    // Geometric and Coordinate Transformations
    node_F_VN_CalibrateCamera : Node_F_VN_CalibrateCamera;
    //node_F_VN_CalibrateCameraExp : Node_F_VN_CalibrateCameraExp;
    //node_F_VN_CalibrateCameraExp2 : Node_F_VN_CalibrateCameraExp2;
    //node_F_VN_CalibrateCameraExp3 : Node_F_VN_CalibrateCameraExp3;
    //node_F_VN_CalibrateCameraManually : Node_F_VN_CalibrateCameraManually;
    //node_F_VN_CalibrateCameraManuallyExp : Node_F_VN_CalibrateCameraManuallyExp;
    node_F_VN_CalibrateCameraPlanar : Node_F_VN_CalibrateCameraPlanar;
    //node_F_VN_CalibrateCameraPlanarExp : Node_F_VN_CalibrateCameraPlanarExp;
    //node_F_VN_CalibrateLinescanCamera : Node_F_VN_CalibrateLinescanCamera;
    //node_F_VN_CalibrateLinescanCameraExp : Node_F_VN_CalibrateLinescanCamera;
    node_F_VN_CompensateLensDistortion : Node_F_VN_CompensateLensDistortion;
    node_F_VN_CompensateLensDistortionExp1 : Node_F_VN_CompensateLensDistortionExp1;
    node_F_VN_CompensateLensDistortionExp2 : Node_F_VN_CompensateLensDistortionExp2;
    node_F_VN_CompensateLensDistortionForPoints : Node_F_VN_CompensateLensDistortionForPoints;
    node_F_VN_CompensateLensDistortionForPointsExp1 : Node_F_VN_CompensateLensDistortionForPointsExp1;
    node_F_VN_CompensateLensDistortionForPointsExp2 : Node_F_VN_CompensateLensDistortionForPointsExp2;
    node_F_VN_DetectPatternPoints : Node_F_VN_DetectPatternPoints;
    //node_F_VN_DetectPatternPointsExp : Node_F_VN_DetectPatternPointsExp;
    node_F_VN_GenerateCalibrationPatternReferencePoints : Node_F_VN_GenerateCalibrationPatternReferencePoints;
    //node_F_VN_ImagePointsWorldDistance : Node_F_VN_ImagePointsWorldDistance;
    node_F_VN_SolvePnP : Node_F_VN_SolvePnP;
    node_F_VN_SolvePnPExp : Node_F_VN_SolvePnPExp;
    node_F_VN_SortDetectedPatternPoints : Node_F_VN_SortDetectedPatternPoints;
    //node_F_VN_TransformCoordinatesImageToWorld_Container : Node_F_VN_TransformCoordinatesImageToWorld_Container;
    //node_F_VN_TransformCoordinatesImageToWorld_Point : Node_F_VN_TransformCoordinatesImageToWorld_Point;
    //node_F_VN_TransformCoordinatesPlanar_Container : Node_F_VN_TransformCoordinatesPlanar_Container;
    //node_F_VN_TransformCoordinatesPlanar_Point : Node_F_VN_TransformCoordinatesPlanar_Point;
    //node_F_VN_TransformCoordinatesWorldToImage_Container : Node_F_VN_TransformCoordinatesWorldToImage_Container;
    //node_F_VN_TransformCoordinatesWorldToImage_Point : Node_F_VN_TransformCoordinatesWorldToImage_Point;
    node_F_VN_AlignRotatedImageRegion : Node_F_VN_AlignRotatedImageRegion;
    node_F_VN_AlignRotatedImageRegionExp : Node_F_VN_AlignRotatedImageRegionExp;
    node_F_VN_ApplyRotationToAffineTransformation : Node_F_VN_ApplyRotationToAffineTransformation;
    node_F_VN_ApplyRotationToAffineTransformationExp : Node_F_VN_ApplyRotationToAffineTransformationExp;
    node_F_VN_ApplyScalingToAffineTransformation : Node_F_VN_ApplyScalingToAffineTransformation;
    node_F_VN_ApplyScalingToAffineTransformationExp : Node_F_VN_ApplyScalingToAffineTransformationExp;
    node_F_VN_ApplyTranslationToAffineTransformation : Node_F_VN_ApplyTranslationToAffineTransformation;
    node_F_VN_ApplyTranslationToAffineTransformationExp : Node_F_VN_ApplyTranslationToAffineTransformationExp;
    node_F_VN_ApplyYAxisInversionToAffineTransformation : Node_F_VN_ApplyYAxisInversionToAffineTransformation;
    node_F_VN_ApplyYAxisInversionToAffineTransformationExp : Node_F_VN_ApplyYAxisInversionToAffineTransformationExp;
    // Polarization
    node_F_VN_DemosaicPolarizedImage : Node_F_VN_DemosaicPolarizedImage;
    node_F_VN_AngleAndDegreeOfLinearPolarization : Node_F_VN_AngleAndDegreeOfLinearPolarization;
    node_F_VN_PolarizedImageGlareReduction : Node_F_VN_PolarizedImageGlareReduction;
    node_F_VN_ConvertCartesianToPolarAngleImage : Node_F_VN_ConvertCartesianToPolarAngleImage;
    node_F_VN_ConvertCartesianToPolarAngleImageExp : Node_F_VN_ConvertCartesianToPolarAngleImageExp;
    node_F_VN_ConvertCartesianToPolarAngles : Node_F_VN_ConvertCartesianToPolarAngles;
    node_F_VN_ConvertCartesianToPolarAnglesExp : Node_F_VN_ConvertCartesianToPolarAnglesExp;
    node_F_VN_ConvertCartesianToPolarImages : Node_F_VN_ConvertCartesianToPolarImages;
    node_F_VN_ConvertCartesianToPolarImagesExp : Node_F_VN_ConvertCartesianToPolarImagesExp;
    node_F_VN_ConvertCartesianToPolarMagnitudeImage : Node_F_VN_ConvertCartesianToPolarMagnitudeImage;
    node_F_VN_ConvertCartesianToPolarMagnitudes : Node_F_VN_ConvertCartesianToPolarMagnitudes;
    node_F_VN_ConvertCartesianToPolarPoints : Node_F_VN_ConvertCartesianToPolarPoints;
    node_F_VN_ConvertCartesianToPolarPointsExp : Node_F_VN_ConvertCartesianToPolarPointsExp;
    node_F_VN_ConvertPolarToCartesianImages : Node_F_VN_ConvertPolarToCartesianImages;
    node_F_VN_ConvertPolarToCartesianImagesExp : Node_F_VN_ConvertPolarToCartesianImagesExp;
    node_F_VN_ConvertPolarToCartesianPoints : Node_F_VN_ConvertPolarToCartesianPoints;
    node_F_VN_ConvertPolarToCartesianPointsExp : Node_F_VN_ConvertPolarToCartesianPointsExp;
    //node_F_VN_DecomposeAffineTransformation : F_VN_DecomposeAffineTransformation;
    node_F_VN_DecomposeAffineTransformation : Node_F_VN_DecomposeAffineTransformation;
    node_F_VN_DecomposeAffineTransformationExp : Node_F_VN_DecomposeAffineTransformationExp;
    //node_F_VN_DecomposeHomography : Node_F_VN_DecomposeHomography;
    //node_F_VN_DecomposeHomographyExp : Node_F_VN_DecomposeHomographyExp;
    node_F_VN_FlipImage : Node_F_VN_FlipImage;
    node_F_VN_GenerateAffineTransformationUnitMatrix2D : Node_F_VN_GenerateAffineTransformationUnitMatrix2D;
    node_F_VN_GetAffineTransformation : Node_F_VN_GetAffineTransformation;
    node_F_VN_GetAffineTransformation2D : Node_F_VN_GetAffineTransformation2D;
    //node_F_VN_GetAffineTransformation2DExp : Node_F_VN_GetAffineTransformation2DExp;
    node_F_VN_GetPerspectiveTransformation : Node_F_VN_GetPerspectiveTransformation;
    node_F_VN_Homography : Node_F_VN_Homography;
    node_F_VN_HomographyExp : Node_F_VN_HomographyExp;
    node_F_VN_InvertAffineTransformation : Node_F_VN_InvertAffineTransformation;
    node_F_VN_PerspectiveTransformation : Node_F_VN_PerspectiveTransformation;
    node_F_VN_PyramidDown : Node_F_VN_PyramidDown;
    node_F_VN_PyramidUp : Node_F_VN_PyramidUp;
    node_F_VN_ConvertMaps : Node_F_VN_ConvertMaps;
    node_F_VN_RemapImage : Node_F_VN_RemapImage;
    node_F_VN_RemapImageExp : Node_F_VN_RemapImageExp;
    node_F_VN_RemapImageToLogPolarSpace : Node_F_VN_RemapImageToLogPolarSpace;
    node_F_VN_RemapImageToLogPolarSpaceExp : Node_F_VN_RemapImageToLogPolarSpaceExp;
    node_F_VN_RemapImageToLogPolarSpaceExp2 : Node_F_VN_RemapImageToLogPolarSpaceExp2;
    node_F_VN_RemapImageToPolarSpace : Node_F_VN_RemapImageToPolarSpace;
    node_F_VN_RemapImageToPolarSpaceExp : Node_F_VN_RemapImageToPolarSpaceExp;
    node_F_VN_RemapImageToPolarSpaceExp2 : Node_F_VN_RemapImageToPolarSpaceExp2;
    node_F_VN_ResizeImage : Node_F_VN_ResizeImage;
    node_F_VN_ResizeImageExp : Node_F_VN_ResizeImageExp;
	node_F_VN_ResizeRegion_TcVnRectangle_DINT : Node_F_VN_ResizeRegion_TcVnRectangle_DINT;
    node_F_VN_RotateImage : Node_F_VN_RotateImage;
    node_F_VN_RotateImageExp : Node_F_VN_RotateImageExp;
    node_F_VN_RotateImageExp2 : Node_F_VN_RotateImageExp2;
    node_F_VN_WarpAffine : Node_F_VN_WarpAffine;
    node_F_VN_WarpAffine_Container : Node_F_VN_WarpAffine_Container;
    node_F_VN_WarpAffine_Point : Node_F_VN_WarpAffine_Point;
    node_F_VN_WarpAffine_Rectangle : Node_F_VN_WarpAffine_Rectangle;
    node_F_VN_WarpAffineExp : Node_F_VN_WarpAffineExp;
    node_F_VN_WarpPerspective : Node_F_VN_WarpPerspective;
    node_F_VN_WarpPerspective_Container : Node_F_VN_WarpPerspective_Container;
    node_F_VN_WarpPerspective_Point : Node_F_VN_WarpPerspective_Point;
    node_F_VN_WarpPerspective_Rectangle : Node_F_VN_WarpPerspective_Rectangle;
    node_F_VN_WarpPerspectiveExp : Node_F_VN_WarpPerspectiveExp;
    
	// Helpers
	node_Mux10Way_ITcVnImage : Node_Mux10Way_ITcVnImage;
	
    // Image Analysis
    //node_F_VN_AdjustActiveContour : Node_F_VN_AdjustActiveContour;
    node_F_VN_SalientFeatures : Node_F_VN_SalientFeatures;
    node_F_VN_FindRois : Node_F_VN_FindRois;
    node_F_VN_MergeRegions : Node_F_VN_MergeRegions;
    node_F_VN_DetectBlobs : Node_F_VN_DetectBlobs;
    node_F_VN_DetectBlobsExp : Node_F_VN_DetectBlobsExp;
    node_F_VN_FindContourHierarchyExp : Node_F_VN_FindContourHierarchyExp;
    node_F_VN_FindContours : Node_F_VN_FindContours;
    node_F_VN_FindContoursExp : Node_F_VN_FindContoursExp;
	node_F_VN_FindTemplateWalsh : Node_F_VN_FindTemplateWalsh;
	node_F_VN_FindTemplateWalsh_AngleRange : Node_F_VN_FindTemplateWalsh_AngleRange;
	node_F_VN_FindTemplateWalshExp : Node_F_VN_FindTemplateWalshExp;
	node_F_VN_FindTemplateWalshExp_AngleRange : Node_F_VN_FindTemplateWalshExp_AngleRange;
    node_F_VN_HoughCircles : Node_F_VN_HoughCircles;
    node_F_VN_HoughCirclesExp : Node_F_VN_HoughCirclesExp;
    node_F_VN_HoughLines : Node_F_VN_HoughLines;
    //node_F_VN_HoughLinesExp : Node_F_VN_HoughLinesExp;
    node_F_VN_HoughLinesP : Node_F_VN_HoughLinesP;
    node_F_VN_HoughLinesPExp : Node_F_VN_HoughLinesPExp;
    node_F_VN_MatchImageHuMoments : Node_F_VN_MatchImageHuMoments;
    node_F_VN_MatchTemplate : Node_F_VN_MatchTemplate;
    node_F_VN_MatchTemplateAndEvaluate : Node_F_VN_MatchTemplateAndEvaluate;
	node_F_VN_MatchTemplateWalsh : Node_F_VN_MatchTemplateWalsh;
	node_F_VN_MatchTemplateWalshExp : Node_F_VN_MatchTemplateWalshExp;
    node_F_VN_MatchTemplateAndEvaluateExp : Node_F_VN_MatchTemplateAndEvaluateExp;
    node_F_VN_MatchTemplateExp : Node_F_VN_MatchTemplateExp;
    node_F_VN_CannyEdgeDetection : Node_F_VN_CannyEdgeDetection;
    node_F_VN_CannyEdgeDetectionExp : Node_F_VN_CannyEdgeDetectionExp;
    node_F_VN_ConnectedComponents : Node_F_VN_ConnectedComponents;
    node_F_VN_ConnectedComponentsExp : Node_F_VN_ConnectedComponentsExp;
    node_F_VN_ConnectedComponentsWithStats : Node_F_VN_ConnectedComponentsWithStats;
    node_F_VN_ConnectedComponentsWithStatsExp : Node_F_VN_ConnectedComponentsWithStatsExp;
    node_F_VN_CountNonZeroPixels : Node_F_VN_CountNonZeroPixels;
    node_F_VN_DistanceTransformation : Node_F_VN_DistanceTransformation;
    node_F_VN_DistanceTransformationExp : Node_F_VN_DistanceTransformationExp;
    node_F_VN_GetConnectedComponent : Node_F_VN_GetConnectedComponent;
    node_F_VN_GetConnectedComponentExp : Node_F_VN_GetConnectedComponentExp;
    node_F_VN_ImageAverage : Node_F_VN_ImageAverage;
    node_F_VN_ImageAverageExp : Node_F_VN_ImageAverageExp;
    node_F_VN_ImageAverageStdDev : Node_F_VN_ImageAverageStdDev;
    node_F_VN_ImageAverageStdDevExp : Node_F_VN_ImageAverageStdDevExp;
    node_F_VN_ImageCenterOfMass : Node_F_VN_ImageCenterOfMass;
    node_F_VN_ImageCenterOfMassExp : Node_F_VN_ImageCenterOfMassExp;
    node_F_VN_ImageMedian : Node_F_VN_ImageMedian;
    node_F_VN_ImageMedianExp : Node_F_VN_ImageMedianExp;
    node_F_VN_ImageMoments : Node_F_VN_ImageMoments;
    node_F_VN_MaxPixelValue : Node_F_VN_MaxPixelValue;
    node_F_VN_MaxPixelValueExp : Node_F_VN_MaxPixelValueExp;
    node_F_VN_MinPixelValue : Node_F_VN_MinPixelValue;
    node_F_VN_MinPixelValueExp : Node_F_VN_MinPixelValueExp;
    node_F_VN_RegionOrientation : Node_F_VN_RegionOrientation;
    node_F_VN_RegionOrientationExp : Node_F_VN_RegionOrientationExp;
    node_F_VN_ImageAbsoluteAverage : Node_F_VN_ImageAbsoluteAverage;
    node_F_VN_UprightInnerRectangle : Node_F_VN_UprightInnerRectangle;
    node_F_VN_UprightInnerRectangleExp : Node_F_VN_UprightInnerRectangleExp;
    
    // Image Color and Contrast Processing
    node_F_VN_ApplyColorMap : Node_F_VN_ApplyColorMap;
    //node_F_VN_ApplyLut : Node_F_VN_ApplyLut;
    node_F_VN_Clahe : Node_F_VN_Clahe;
    node_F_VN_ClaheExp : Node_F_VN_ClaheExp;
    node_F_VN_ConvertColorSpace : Node_F_VN_ConvertColorSpace;
    node_F_VN_GenerateColorMap : Node_F_VN_GenerateColorMap;
    node_F_VN_GenerateCustomColorMap : Node_F_VN_GenerateCustomColorMap;
    node_F_VN_Histogram : Node_F_VN_Histogram;
    node_F_VN_HistogramEqualization : Node_F_VN_HistogramEqualization;
    node_F_VN_HistogramEqualizationExp : Node_F_VN_HistogramEqualizationExp;
	node_F_VN_HistogramExp : Node_F_VN_HistogramExp;
    node_F_VN_InvertImageColor : Node_F_VN_InvertImageColor;
    node_F_VN_InvertImageColorExp : Node_F_VN_InvertImageColorExp;
    node_F_VN_NormalizeImage : Node_F_VN_NormalizeImage;
    node_F_VN_NormalizeImageExp : Node_F_VN_NormalizeImageExp;
    node_F_VN_NormalizeImageForDisplay : Node_F_VN_NormalizeImageForDisplay;
    //node_F_VN_ReferenceColorSimilarity_ITcVnColorModel : Node_F_VN_ReferenceColorSimilarity_ITcVnColorModel;
    //node_F_VN_ReferenceColorSimilarity_ITcVnMlModel : Node_F_VN_ReferenceColorSimilarity_ITcVnMlModel;
    node_F_VN_ReferenceColorSimilarity_TcVnVector3_LREAL : Node_F_VN_ReferenceColorSimilarity_TcVnVector3_LREAL;
    //node_F_VN_ReferenceColorSimilarityExp_ITcVnColorModel : Node_F_VN_ReferenceColorSimilarityExp_ITcVnColorModel;
    //node_F_VN_ReferenceColorSimilarityExp_ITcVnColorModel : Node_F_VN_ReferenceColorSimilarityExp_ITcVnColorModel;
    node_F_VN_ReferenceColorSimilarityExp_TcVnVector3_LREAL : Node_F_VN_ReferenceColorSimilarityExp_TcVnVector3_LREAL;
    //node_F_VN_TrainImageColor : Node_F_VN_TrainImageColor;
    //node_F_VN_TrainImageColor_ITcVnMlModel : Node_F_VN_TrainImageColor_ITcVnMlModel;
    //node_F_VN_TrainImageColorExp : Node_F_VN_TrainImageColorExp;
    //node_F_VN_TrainImageColorExp_ITcVnMlModel : Node_F_VN_TrainImageColorExp_ITcVnMlModel;
    //node_F_VN_TrainImageColorExp2 : Node_F_VN_TrainImageColorExp2;
    //node_F_VN_TrainImageColorExp2_ITcVnMlModel : Node_F_VN_TrainImageColorExp2_ITcVnMlModel;
    node_F_VN_WhiteBalance : Node_F_VN_WhiteBalance;
    
    // Image Filtering
    node_F_VN_BilateralFilter : Node_F_VN_BilateralFilter;
    node_F_VN_BilateralFilterExp : Node_F_VN_BilateralFilterExp;
    node_F_VN_BoxFilter : Node_F_VN_BoxFilter;
    node_F_VN_BoxFilterExp : Node_F_VN_BoxFilterExp;
    node_F_VN_BrightBorderObjects : Node_F_VN_BrightBorderObjects;
    node_F_VN_CreateStructuringElement : Node_F_VN_CreateStructuringElement;
    //node_F_VN_CustomFilter : Node_F_VN_CustomFilter;
    //node_F_VN_CustomFilterExp : Node_F_VN_CustomFilterExp;
    node_F_VN_DarkBorderObjects : Node_F_VN_DarkBorderObjects;
    node_F_VN_FillHoles : Node_F_VN_FillHoles;
    node_F_VN_GaussianFilter : Node_F_VN_GaussianFilter;
    node_F_VN_GaussianFilterExp : Node_F_VN_GaussianFilterExp;
    node_F_VN_LaplacianFilter : Node_F_VN_LaplacianFilter;
    node_F_VN_LaplacianFilterExp : Node_F_VN_LaplacianFilterExp;
    node_F_VN_LocalMaxima : Node_F_VN_LocalMaxima;
    node_F_VN_LocalMinima : Node_F_VN_LocalMinima;
    node_F_VN_MedianFilter : Node_F_VN_MedianFilter;
    node_F_VN_MorphologicalOperator : Node_F_VN_MorphologicalOperator;
    node_F_VN_RemoveLocalMaxima : Node_F_VN_RemoveLocalMaxima;
    node_F_VN_RemoveLocalMinima : Node_F_VN_RemoveLocalMinima;
    node_F_VN_ScharrFilter : Node_F_VN_ScharrFilter;
    node_F_VN_ScharrFilterExp : Node_F_VN_ScharrFilterExp;
    //node_F_VN_SeparableCustomFilter : Node_F_VN_SeparableCustomFilter;
    //node_F_VN_SeparableCustomFilterExp : Node_F_VN_SeparableCustomFilterExp;
    node_F_VN_SobelFilter : Node_F_VN_SobelFilter;
    node_F_VN_SobelFilterExp : Node_F_VN_SobelFilterExp;
    node_F_VN_VarianceFilter : Node_F_VN_VarianceFilter;
    node_F_VN_VarianceFilterExp : Node_F_VN_VarianceFilterExp;
    
    // Image Segmentation
    node_F_VN_AdaptiveThreshold : Node_F_VN_AdaptiveThreshold;
    node_F_VN_AdaptiveThresholdExp : Node_F_VN_AdaptiveThresholdExp;
    node_F_VN_CheckColorRange : Node_F_VN_CheckColorRange;
    node_F_VN_DoubleThreshold : Node_F_VN_DoubleThreshold;
    node_F_VN_Threshold : Node_F_VN_Threshold;
    node_F_VN_WatershedSegmentationExp : Node_F_VN_WatershedSegmentationExp;
    node_F_VN_SauvolaThreshold : Node_F_VN_SauvolaThreshold;
    
    // Keypoint Features
    node_F_VN_FilterGoodMatches : Node_F_VN_FilterGoodMatches;
    node_F_VN_FindReferenceKeyPointsInImage : Node_F_VN_FindReferenceKeyPointsInImage;
    node_F_VN_FindReferenceKeyPointsInImageAKAZE : Node_F_VN_FindReferenceKeyPointsInImageAKAZE;
    node_F_VN_FindReferenceKeyPointsInImageAKAZEExp : Node_F_VN_FindReferenceKeyPointsInImageAKAZEExp;
    node_F_VN_FindReferenceKeyPointsInImageBRISK : Node_F_VN_FindReferenceKeyPointsInImageBRISK;
    node_F_VN_FindReferenceKeyPointsInImageBRISKExp : Node_F_VN_FindReferenceKeyPointsInImageBRISKExp;
    node_F_VN_FindReferenceKeyPointsInImageExp : Node_F_VN_FindReferenceKeyPointsInImageExp;
    node_F_VN_FindReferenceKeyPointsInImageORB : Node_F_VN_FindReferenceKeyPointsInImageORB;
    node_F_VN_FindReferenceKeyPointsInImageORBExp : Node_F_VN_FindReferenceKeyPointsInImageORBExp;
    node_F_VN_GetMatchCoordinates : Node_F_VN_GetMatchCoordinates;
    node_F_VN_KeyPointsAGAST : Node_F_VN_KeyPointsAGAST;
    node_F_VN_KeyPointsAGASTExp : Node_F_VN_KeyPointsAGASTExp;
    node_F_VN_KeyPointsAndDescriptorsAKAZE : Node_F_VN_KeyPointsAndDescriptorsAKAZE;
    node_F_VN_KeyPointsAndDescriptorsAKAZEExp : Node_F_VN_KeyPointsAndDescriptorsAKAZEExp;
    node_F_VN_KeyPointsAndDescriptorsBRISK : Node_F_VN_KeyPointsAndDescriptorsBRISK;
    node_F_VN_KeyPointsAndDescriptorsBRISKExp : Node_F_VN_KeyPointsAndDescriptorsBRISKExp;
    node_F_VN_KeyPointsAndDescriptorsKAZE : Node_F_VN_KeyPointsAndDescriptorsKAZE;
    node_F_VN_KeyPointsAndDescriptorsKAZEExp : Node_F_VN_KeyPointsAndDescriptorsKAZEExp;
    node_F_VN_KeyPointsAndDescriptorsORB : Node_F_VN_KeyPointsAndDescriptorsORB;
    node_F_VN_KeyPointsAndDescriptorsORBExp : Node_F_VN_KeyPointsAndDescriptorsORBExp;
    node_F_VN_KeyPointsFAST : Node_F_VN_KeyPointsFAST;
    node_F_VN_KeyPointsFASTExp : Node_F_VN_KeyPointsFASTExp;
    node_F_VN_KeyPointsGFTT : Node_F_VN_KeyPointsGFTT;
    node_F_VN_KeyPointsGFTTExp : Node_F_VN_KeyPointsGFTTExp;
    node_F_VN_KeyPointsMSER : Node_F_VN_KeyPointsMSER;
    node_F_VN_KeyPointsMSERExp : Node_F_VN_KeyPointsMSERExp;
    node_F_VN_KeyPointsSB : Node_F_VN_KeyPointsSB;
    node_F_VN_KeyPointsSBExp : Node_F_VN_KeyPointsSBExp;
    node_F_VN_MatchDescriptorsBF : Node_F_VN_MatchDescriptorsBF;
    node_F_VN_MatchDescriptorsBFExp : Node_F_VN_MatchDescriptorsBFExp;
    node_F_VN_MatchDescriptorsFlannLsh : Node_F_VN_MatchDescriptorsFlannLsh;
    node_F_VN_MatchDescriptorsFlannLshExp : Node_F_VN_MatchDescriptorsFlannLshExp;
    node_F_VN_MatchDescriptorsKnnBF : Node_F_VN_MatchDescriptorsKnnBF;
    node_F_VN_MatchDescriptorsKnnBFExp : Node_F_VN_MatchDescriptorsKnnBFExp;
    node_F_VN_MatchDescriptorsKnnFlannLsh : Node_F_VN_MatchDescriptorsKnnFlannLsh;
    node_F_VN_MatchDescriptorsKnnFlannLshExp : Node_F_VN_MatchDescriptorsKnnFlannLshExp;
    node_F_VN_RegionsMSER : Node_F_VN_RegionsMSER;
    node_F_VN_RegionsMSERExp : Node_F_VN_RegionsMSERExp;
    
    // Machine Learning
    //node_F_VN_CreateBoostClassifier : Node_F_VN_CreateBoostClassifier;
    //node_F_VN_CreateBoostClassifierExp : Node_F_VN_CreateBoostClassifierExp;
    //node_F_VN_CreateBoostClassifierExp2 : Node_F_VN_CreateBoostClassifierExp2;
    //node_F_VN_CreateKmppModel : Node_F_VN_CreateKmppModel;
    //node_F_VN_CreateKmppModelExp : Node_F_VN_CreateKmppModelExp;
    //node_F_VN_CreateKnnModel : Node_F_VN_CreateKnnModel;
    //node_F_VN_CreateLbgModel : Node_F_VN_CreateLbgModel;
    //node_F_VN_CreateLbgModelExp : Node_F_VN_CreateLbgModelExp;
    //node_F_VN_CreateLdaTransform : Node_F_VN_CreateLdaTransform;
    //node_F_VN_CreateLdaTransformViaComponentNum : Node_F_VN_CreateLdaTransformViaComponentNum;
    //node_F_VN_CreateNbcModel : Node_F_VN_CreateNbcModel;
    //node_F_VN_CreatePcaTransform : Node_F_VN_CreatePcaTransform;
    //node_F_VN_CreatePcaTransformViaComponentNum : Node_F_VN_CreatePcaTransformViaComponentNum;
    //node_F_VN_CreatePcaTransformViaVariance : Node_F_VN_CreatePcaTransformViaVariance;
    //node_F_VN_CreateRTreesModel : Node_F_VN_CreateRTreesModel;
    //node_F_VN_CreateRTreesModelExp : Node_F_VN_CreateRTreesModelExp;
    //node_F_VN_CreateRTreesModelExp2 : Node_F_VN_CreateRTreesModelExp2;
    //node_F_VN_CreateStaModel : Node_F_VN_CreateStaModel;
    //node_F_VN_CreateStaModelExp : Node_F_VN_CreateStaModelExp;
    //node_F_VN_CreateStaModelExp2 : Node_F_VN_CreateStaModelExp2;
    //node_F_VN_CreateSvmModel : Node_F_VN_CreateSvmModel;
    //node_F_VN_CreateSvmModelExp : Node_F_VN_CreateSvmModelExp;
    //node_F_VN_CreateSvmModelExp2 : Node_F_VN_CreateSvmModelExp2;
    //node_F_VN_CreateSvmSgdClassifier : Node_F_VN_CreateSvmSgdClassifier;
    //node_F_VN_CreateSvmSgdClassifierExp : Node_F_VN_CreateSvmSgdClassifierExp;
    //node_F_VN_FeatureScaling : Node_F_VN_FeatureScaling;
    //node_F_VN_FeatureScalingExp : Node_F_VN_FeatureScalingExp;
    //node_F_VN_FeatureTransform : Node_F_VN_FeatureTransform;
    //node_F_VN_GetBatchClusters : Node_F_VN_GetBatchClusters;
    //node_F_VN_GetBatchClustersExp : Node_F_VN_GetBatchClustersExp;
    //node_F_VN_GetBatchNovelties : Node_F_VN_GetBatchNovelties;
    //node_F_VN_GetClusterCenter : Node_F_VN_GetClusterCenter;
    //node_F_VN_GetClusterNum : Node_F_VN_GetClusterNum;
    //node_F_VN_GetFeatureScales : Node_F_VN_GetFeatureScales;
    //node_F_VN_GetSampleCluster : Node_F_VN_GetSampleCluster;
    //node_F_VN_GetSampleClusterExp : Node_F_VN_GetSampleClusterExp;
    //node_F_VN_GetSampleNovelty : Node_F_VN_GetSampleNovelty;
    //node_F_VN_InverseFeatureScaling : Node_F_VN_InverseFeatureScaling;
    //node_F_VN_InverseFeatureScaling_REAL : Node_F_VN_InverseFeatureScaling_REAL;
    //node_F_VN_InverseFeatureScalingExp : Node_F_VN_InverseFeatureScalingExp;
    //node_F_VN_InverseFeatureScalingExp_REAL : Node_F_VN_InverseFeatureScalingExp_REAL;
    //node_F_VN_InverseFeatureTransform : Node_F_VN_InverseFeatureTransform;
    //node_F_VN_PredictBatch : Node_F_VN_PredictBatch;
    //node_F_VN_PredictBatchExp : Node_F_VN_PredictBatchExp;
    //node_F_VN_PredictSampleClass : Node_F_VN_PredictSampleClass;
    //node_F_VN_PredictSampleClassExp : Node_F_VN_PredictSampleClassExp;
    //node_F_VN_PredictSampleScalar : Node_F_VN_PredictSampleScalar;
    //node_F_VN_PredictSampleScalarExp : Node_F_VN_PredictSampleScalarExp;
    //node_F_VN_PredictSampleVector : Node_F_VN_PredictSampleVector;
    //node_F_VN_PredictSampleVectorExp : Node_F_VN_PredictSampleVectorExp;
    //node_F_VN_TrainBatch : Node_F_VN_TrainBatch;
    //node_F_VN_TrainBatchClusters : Node_F_VN_TrainBatchClusters;
    //node_F_VN_TrainSample : Node_F_VN_TrainSample;
    //node_F_VN_TrainSampleClass : Node_F_VN_TrainSampleClass;
    //node_F_VN_TrainSampleCluster : Node_F_VN_TrainSampleCluster;
    //node_F_VN_TrainSampleScalar : Node_F_VN_TrainSampleScalar;
    //node_F_VN_TrainSampleVector : Node_F_VN_TrainSampleVector;

    // Measurement
    node_F_VN_AdjustSearchWindowOrientationToLinearEdge : Node_F_VN_AdjustSearchWindowOrientationToLinearEdge;
	node_F_VN_ClosestPointsBF : Node_F_VN_ClosestPointsBF;
    node_F_VN_LocateAxisAlignedEdges : Node_F_VN_LocateAxisAlignedEdges;
    node_F_VN_LocateAxisAlignedEdgesExp : Node_F_VN_LocateAxisAlignedEdgesExp;
	node_F_VN_LocateCircularArc : Node_F_VN_LocateCircularArc;
    node_F_VN_LocateCircularArcExp : Node_F_VN_LocateCircularArcExp;
    node_F_VN_LocateCircularArcExp2 : Node_F_VN_LocateCircularArcExp2;
    node_F_VN_LocateEdge : Node_F_VN_LocateEdge;
    node_F_VN_LocateEdgeExp : Node_F_VN_LocateEdgeExp;
    node_F_VN_LocateEdgeExp2 : Node_F_VN_LocateEdgeExp2;
    node_F_VN_LocateEdges : Node_F_VN_LocateEdges;
    node_F_VN_LocateEdgesExp : Node_F_VN_LocateEdgesExp;
    node_F_VN_LocateEdgesExp2 : Node_F_VN_LocateEdgesExp2;
    node_F_VN_LocateEllipse : Node_F_VN_LocateEllipse;
	node_F_VN_LocateEllipseExp : Node_F_VN_LocateEllipseExp;
    node_F_VN_LocateEllipseExp2 : Node_F_VN_LocateEllipseExp2;
    node_F_VN_MeasureAngleBetweenEdges : Node_F_VN_MeasureAngleBetweenEdges;
    node_F_VN_MeasureAngleBetweenEdgesExp : Node_F_VN_MeasureAngleBetweenEdgesExp;
    node_F_VN_MeasureAngleBetweenEdgesExp2 : Node_F_VN_MeasureAngleBetweenEdgesExp2;
    node_F_VN_MeasureEdgeDistance : Node_F_VN_MeasureEdgeDistance;
	node_F_VN_MeasureEdgeDistanceExp : Node_F_VN_MeasureEdgeDistanceExp;
    node_F_VN_MeasureEdgeDistanceExp2 : Node_F_VN_MeasureEdgeDistanceExp2;
    node_F_VN_MeasureMinEdgeDistance : Node_F_VN_MeasureMinEdgeDistance;
    node_F_VN_MeasureMinEdgeDistanceExp : Node_F_VN_MeasureMinEdgeDistanceExp;
    node_F_VN_MeasureMinEdgeDistanceExp2 : Node_F_VN_MeasureMinEdgeDistanceExp2;
    
    // Miscellaneous
    node_F_VN_CheckFunctionInitialization : Node_F_VN_CheckFunctionInitialization;
    node_F_VN_ClipLineToBoundary : Node_F_VN_ClipLineToBoundary;
    node_F_VN_ClipLineToBoundary_ITcVnImage : Node_F_VN_ClipLineToBoundary_ITcVnImage;
    node_F_VN_ClipLineToBoundary_TcVnRectangle_DINT : Node_F_VN_ClipLineToBoundary_TcVnRectangle_DINT;
    //node_F_VN_ConvertITcUnknownToITcVnBitmapExport : Node_F_VN_ConvertITcUnknownToITcVnBitmapExport;
    //node_F_VN_ConvertITcUnknownToITcVnContainer : Node_F_VN_ConvertITcUnknownToITcVnContainer;
    //node_F_VN_ConvertITcUnknownToITcVnImage : Node_F_VN_ConvertITcUnknownToITcVnImage;
    //node_F_VN_ConvertITcUnknownToITcVnMlModel : Node_F_VN_ConvertITcUnknownToITcVnMlModel;
    node_F_VN_DeinitializeFunction : Node_F_VN_DeinitializeFunction;
    //node_F_VN_GetTimestamp : Node_F_VN_GetTimestamp;
    node_F_VN_HuMomentInvariants : Node_F_VN_HuMomentInvariants;
    //node_F_VN_InitMatrixStruct : Node_F_VN_InitMatrixStruct;
    node_F_VN_InvertMatrix3x3 : Node_F_VN_InvertMatrix3x3;
    node_F_VN_LineIntersectionPoint : Node_F_VN_LineIntersectionPoint;
    node_F_VN_LineIntersectionPointAndAngle : Node_F_VN_LineIntersectionPointAndAngle;
    //node_F_VN_MultiplyMatrices : Node_F_VN_MultiplyMatrices;
    node_F_VN_OrthogonalVector_TcVnVector2_DINT : Node_F_VN_OrthogonalVector_TcVnVector2_DINT;
    node_F_VN_OrthogonalVector_TcVnVector2_LREAL : Node_F_VN_OrthogonalVector_TcVnVector2_LREAL;
    node_F_VN_OrthogonalVector_TcVnVector2_REAL : Node_F_VN_OrthogonalVector_TcVnVector2_REAL;
    node_F_VN_PointToLineDistance_TcVnPoint2_DINT : Node_F_VN_PointToLineDistance_TcVnPoint2_DINT;
    node_F_VN_PointToLineDistance_TcVnPoint2_LREAL : Node_F_VN_PointToLineDistance_TcVnPoint2_LREAL;
    node_F_VN_PointToLineDistance_TcVnPoint2_REAL : Node_F_VN_PointToLineDistance_TcVnPoint2_REAL;
    node_F_VN_PointToPointDirection_TcVnPoint2_DINT : Node_F_VN_PointToPointDirection_TcVnPoint2_DINT;
    node_F_VN_PointToPointDirection_TcVnPoint2_LREAL : Node_F_VN_PointToPointDirection_TcVnPoint2_LREAL;
    node_F_VN_PointToPointDirection_TcVnPoint2_REAL : Node_F_VN_PointToPointDirection_TcVnPoint2_REAL;
    node_F_VN_PointToPointDistance_TcVnPoint2_DINT : Node_F_VN_PointToPointDistance_TcVnPoint2_DINT;
    node_F_VN_PointToPointDistance_TcVnPoint2_LREAL : Node_F_VN_PointToPointDistance_TcVnPoint2_LREAL;
    node_F_VN_PointToPointDistance_TcVnPoint2_REAL : Node_F_VN_PointToPointDistance_TcVnPoint2_REAL;
    node_F_VN_RotatedRectangleCorners : Node_F_VN_RotatedRectangleCorners;
    node_F_VN_RotatedRectangleIntersection : Node_F_VN_RotatedRectangleIntersection;
    //node_F_VN_SetRngSeed : Node_F_VN_SetRngSeed;
    //node_F_VN_UpdateTimestamp : Node_F_VN_UpdateTimestamp;
    
//     node_FB_VN_InitializeFunction : Node_FB_VN_InitializeFunction;
    
    // OCR
    node_F_VN_OCR : Node_F_VN_OCR;
    node_F_VN_OCRExp : Node_F_VN_OCRExp;
    
    // Texture Analysis
    node_F_VN_Granulometry : Node_F_VN_Granulometry;
    node_F_VN_HaralickFeatures : Node_F_VN_HaralickFeatures;
    
    // Neural Network
    //node_F_VN_ConvertDataLayout : Node_F_VN_ConvertDataLayout;
    //node_F_VN_ExecuteNeuralNetwork : Node_F_VN_ExecuteNeuralNetwork;
    //node_F_VN_ExecuteNeuralNetwork_MultiLayerOutput : Node_F_VN_ExecuteNeuralNetwork_MultiLayerOutput;
    //node_F_VN_ExecuteNeuralNetwork_SingleLayerOutput : Node_F_VN_ExecuteNeuralNetwork_SingleLayerOutput;
    //node_F_VN_GetNeuralNetworkLayerNames : Node_F_VN_GetNeuralNetworkLayerNames;
    //node_F_VN_NonMaxSuppression : Node_F_VN_NonMaxSuppression;
    //node_F_VN_NonMaxSuppressionExp : Node_F_VN_NonMaxSuppressionExp;
	node_F_VN_Reduce : Node_F_VN_Reduce;
	node_F_VN_ReduceArg : Node_F_VN_ReduceArg;
    //node_F_VN_ReshapeImage : Node_F_VN_ReshapeImage;
	node_F_VN_Sigmoid : Node_F_VN_Sigmoid;
	node_F_VN_SigmoidExp : Node_F_VN_SigmoidExp;
	node_F_VN_SoftMax : Node_F_VN_SoftMax;
	
END_VAR

METHOD PUBLIC RegisterWithNodeFactory
VAR_INPUT
	NodeFactory : I_NodeFactory;
END_VAR
// Algebraic Container Operations
NodeFactory.AddNodeAsPrototype('Vision/Algebraic Container Operations/F_VN_AddToContainerElements/F_VN_AddToContainerElements_DINT', node_F_VN_AddToContainerElements_DINT);
NodeFactory.AddNodeAsPrototype('Vision/Algebraic Container Operations/F_VN_AddToContainerElements/F_VN_AddToContainerElements_INT', node_F_VN_AddToContainerElements_INT);
NodeFactory.AddNodeAsPrototype('Vision/Algebraic Container Operations/F_VN_AddToContainerElements/F_VN_AddToContainerElements_LREAL', node_F_VN_AddToContainerElements_LREAL);
NodeFactory.AddNodeAsPrototype('Vision/Algebraic Container Operations/F_VN_AddToContainerElements/F_VN_AddToContainerElements_REAL', node_F_VN_AddToContainerElements_REAL);
NodeFactory.AddNodeAsPrototype('Vision/Algebraic Container Operations/F_VN_AddToContainerElements/F_VN_AddToContainerElements_SINT', node_F_VN_AddToContainerElements_SINT);
NodeFactory.AddNodeAsPrototype('Vision/Algebraic Container Operations/F_VN_AddToContainerElements/F_VN_AddToContainerElements_TcVnKeyPoint', node_F_VN_AddToContainerElements_TcVnKeyPoint);
NodeFactory.AddNodeAsPrototype('Vision/Algebraic Container Operations/F_VN_AddToContainerElements/F_VN_AddToContainerElements_TcVnPoint2_DINT', node_F_VN_AddToContainerElements_TcVnPoint2_DINT);
NodeFactory.AddNodeAsPrototype('Vision/Algebraic Container Operations/F_VN_AddToContainerElements/F_VN_AddToContainerElements_TcVnPoint2_LREAL', node_F_VN_AddToContainerElements_TcVnPoint2_LREAL);
NodeFactory.AddNodeAsPrototype('Vision/Algebraic Container Operations/F_VN_AddToContainerElements/F_VN_AddToContainerElements_TcVnPoint2_REAL', node_F_VN_AddToContainerElements_TcVnPoint2_REAL);
NodeFactory.AddNodeAsPrototype('Vision/Algebraic Container Operations/F_VN_AddToContainerElements/F_VN_AddToContainerElements_TcVnPoint3_LREAL', node_F_VN_AddToContainerElements_TcVnPoint3_LREAL);
NodeFactory.AddNodeAsPrototype('Vision/Algebraic Container Operations/F_VN_AddToContainerElements/F_VN_AddToContainerElements_TcVnPoint3_REAL', node_F_VN_AddToContainerElements_TcVnPoint3_REAL);
NodeFactory.AddNodeAsPrototype('Vision/Algebraic Container Operations/F_VN_AddToContainerElements/F_VN_AddToContainerElements_TcVnRectangle_DINT', node_F_VN_AddToContainerElements_TcVnRectangle_DINT);
NodeFactory.AddNodeAsPrototype('Vision/Algebraic Container Operations/F_VN_AddToContainerElements/F_VN_AddToContainerElements_TcVnRotatedRectangle', node_F_VN_AddToContainerElements_TcVnRotatedRectangle);
NodeFactory.AddNodeAsPrototype('Vision/Algebraic Container Operations/F_VN_AddToContainerElements/F_VN_AddToContainerElements_TcVnVector2_DINT', node_F_VN_AddToContainerElements_TcVnVector2_DINT);
NodeFactory.AddNodeAsPrototype('Vision/Algebraic Container Operations/F_VN_AddToContainerElements/F_VN_AddToContainerElements_TcVnVector2_INT', node_F_VN_AddToContainerElements_TcVnVector2_INT);
NodeFactory.AddNodeAsPrototype('Vision/Algebraic Container Operations/F_VN_AddToContainerElements/F_VN_AddToContainerElements_TcVnVector2_REAL', node_F_VN_AddToContainerElements_TcVnVector2_REAL);
NodeFactory.AddNodeAsPrototype('Vision/Algebraic Container Operations/F_VN_AddToContainerElements/F_VN_AddToContainerElements_TcVnVector2_SINT', node_F_VN_AddToContainerElements_TcVnVector2_SINT);
NodeFactory.AddNodeAsPrototype('Vision/Algebraic Container Operations/F_VN_AddToContainerElements/F_VN_AddToContainerElements_TcVnVector2_UINT', node_F_VN_AddToContainerElements_TcVnVector2_UINT);
NodeFactory.AddNodeAsPrototype('Vision/Algebraic Container Operations/F_VN_AddToContainerElements/F_VN_AddToContainerElements_TcVnVector2_USINT', node_F_VN_AddToContainerElements_TcVnVector2_USINT);
NodeFactory.AddNodeAsPrototype('Vision/Algebraic Container Operations/F_VN_AddToContainerElements/F_VN_AddToContainerElements_TcVnVector3_INT', node_F_VN_AddToContainerElements_TcVnVector3_INT);
NodeFactory.AddNodeAsPrototype('Vision/Algebraic Container Operations/F_VN_AddToContainerElements/F_VN_AddToContainerElements_TcVnVector3_REAL', node_F_VN_AddToContainerElements_TcVnVector3_REAL);
NodeFactory.AddNodeAsPrototype('Vision/Algebraic Container Operations/F_VN_AddToContainerElements/F_VN_AddToContainerElements_TcVnVector3_SINT', node_F_VN_AddToContainerElements_TcVnVector3_SINT);
NodeFactory.AddNodeAsPrototype('Vision/Algebraic Container Operations/F_VN_AddToContainerElements/F_VN_AddToContainerElements_TcVnVector3_UINT', node_F_VN_AddToContainerElements_TcVnVector3_UINT);
NodeFactory.AddNodeAsPrototype('Vision/Algebraic Container Operations/F_VN_AddToContainerElements/F_VN_AddToContainerElements_TcVnVector3_USINT', node_F_VN_AddToContainerElements_TcVnVector3_USINT);
NodeFactory.AddNodeAsPrototype('Vision/Algebraic Container Operations/F_VN_AddToContainerElements/F_VN_AddToContainerElements_TcVnVector4_DINT', node_F_VN_AddToContainerElements_TcVnVector4_DINT);
NodeFactory.AddNodeAsPrototype('Vision/Algebraic Container Operations/F_VN_AddToContainerElements/F_VN_AddToContainerElements_TcVnVector4_INT', node_F_VN_AddToContainerElements_TcVnVector4_INT);
NodeFactory.AddNodeAsPrototype('Vision/Algebraic Container Operations/F_VN_AddToContainerElements/F_VN_AddToContainerElements_TcVnVector4_LREAL', node_F_VN_AddToContainerElements_TcVnVector4_LREAL);
NodeFactory.AddNodeAsPrototype('Vision/Algebraic Container Operations/F_VN_AddToContainerElements/F_VN_AddToContainerElements_TcVnVector4_REAL', node_F_VN_AddToContainerElements_TcVnVector4_REAL);
NodeFactory.AddNodeAsPrototype('Vision/Algebraic Container Operations/F_VN_AddToContainerElements/F_VN_AddToContainerElements_TcVnVector4_SINT', node_F_VN_AddToContainerElements_TcVnVector4_SINT);
NodeFactory.AddNodeAsPrototype('Vision/Algebraic Container Operations/F_VN_AddToContainerElements/F_VN_AddToContainerElements_TcVnVector4_UINT', node_F_VN_AddToContainerElements_TcVnVector4_UINT);
NodeFactory.AddNodeAsPrototype('Vision/Algebraic Container Operations/F_VN_AddToContainerElements/F_VN_AddToContainerElements_TcVnVector4_USINT', node_F_VN_AddToContainerElements_TcVnVector4_USINT);
NodeFactory.AddNodeAsPrototype('Vision/Algebraic Container Operations/F_VN_AddToContainerElements/F_VN_AddToContainerElements_UDINT', node_F_VN_AddToContainerElements_UDINT);
NodeFactory.AddNodeAsPrototype('Vision/Algebraic Container Operations/F_VN_AddToContainerElements/F_VN_AddToContainerElements_UINT', node_F_VN_AddToContainerElements_UINT);
NodeFactory.AddNodeAsPrototype('Vision/Algebraic Container Operations/F_VN_AddToContainerElements/F_VN_AddToContainerElements_ULINT', node_F_VN_AddToContainerElements_ULINT);
NodeFactory.AddNodeAsPrototype('Vision/Algebraic Container Operations/F_VN_AddToContainerElements/F_VN_AddToContainerElements_USINT', node_F_VN_AddToContainerElements_USINT);
NodeFactory.AddNodeAsPrototype('Vision/Algebraic Container Operations/F_VN_AddContainers', node_F_VN_AddContainers);
NodeFactory.AddNodeAsPrototype('Vision/Algebraic Container Operations/F_VN_BitwiseAndContainers', node_F_VN_BitwiseAndContainers);
NodeFactory.AddNodeAsPrototype('Vision/Algebraic Container Operations/F_VN_BitwiseNotContainer', node_F_VN_BitwiseNotContainer);
NodeFactory.AddNodeAsPrototype('Vision/Algebraic Container Operations/F_VN_BitwiseOrContainers', node_F_VN_BitwiseOrContainers);
NodeFactory.AddNodeAsPrototype('Vision/Algebraic Container Operations/F_VN_BitwiseXorContainers', node_F_VN_BitwiseXorContainers);
NodeFactory.AddNodeAsPrototype('Vision/Algebraic Container Operations/F_VN_DivideContainers', node_F_VN_DivideContainers);
NodeFactory.AddNodeAsPrototype('Vision/Algebraic Container Operations/F_VN_DivideContainersExp', node_F_VN_DivideContainersExp);
NodeFactory.AddNodeAsPrototype('Vision/Algebraic Container Operations/F_VN_MaxContainer', node_F_VN_MaxContainer);
NodeFactory.AddNodeAsPrototype('Vision/Algebraic Container Operations/F_VN_MinContainer', node_F_VN_MinContainer);
NodeFactory.AddNodeAsPrototype('Vision/Algebraic Container Operations/F_VN_MultiplyContainers', node_F_VN_MultiplyContainers);
//NodeFactory.AddNodeAsPrototype('Vision/Algebraic Container Operations/F_VN_MultiplyWithContainerElements1', node_F_VN_MultiplyWithContainerElements1);
//NodeFactory.AddNodeAsPrototype('Vision/Algebraic Container Operations/F_VN_MultiplyWithContainerElements2', node_F_VN_MultiplyWithContainerElements2);
//NodeFactory.AddNodeAsPrototype('Vision/Algebraic Container Operations/F_VN_MultiplyWithContainerElements3', node_F_VN_MultiplyWithContainerElements3);
//NodeFactory.AddNodeAsPrototype('Vision/Algebraic Container Operations/F_VN_MultiplyWithContainerElements4', node_F_VN_MultiplyWithContainerElements4);
NodeFactory.AddNodeAsPrototype('Vision/Algebraic Container Operations/F_VN_NegateContainer', node_F_VN_NegateContainer);
NodeFactory.AddNodeAsPrototype('Vision/Algebraic Container Operations/F_VN_SubtractContainers', node_F_VN_SubtractContainers);

// Algebraic Image Operations
NodeFactory.AddNodeAsPrototype('Vision/Algebraic Image Operations/F_VN_AddImages', node_F_VN_AddImages);
NodeFactory.AddNodeAsPrototype('Vision/Algebraic Image Operations/F_VN_AddImagesWeighted', node_F_VN_AddImagesWeighted);
NodeFactory.AddNodeAsPrototype('Vision/Algebraic Image Operations/F_VN_AddImagesWeightedExp', node_F_VN_AddImagesWeightedExp);
NodeFactory.AddNodeAsPrototype('Vision/Algebraic Image Operations/F_VN_AddScalarToImage', node_F_VN_AddScalarToImage);
NodeFactory.AddNodeAsPrototype('Vision/Algebraic Image Operations/F_VN_AddVectorToImage', node_F_VN_AddVectorToImage);
NodeFactory.AddNodeAsPrototype('Vision/Algebraic Image Operations/F_VN_BitwiseAndImages', node_F_VN_BitwiseAndImages);
NodeFactory.AddNodeAsPrototype('Vision/Algebraic Image Operations/F_VN_BitwiseAndImagesExp', node_F_VN_BitwiseAndImagesExp);
NodeFactory.AddNodeAsPrototype('Vision/Algebraic Image Operations/F_VN_BitwiseAndScalarWithImage', node_F_VN_BitwiseAndScalarWithImage);
NodeFactory.AddNodeAsPrototype('Vision/Algebraic Image Operations/F_VN_BitwiseAndVectorWithImage', node_F_VN_BitwiseAndVectorWithImage);
NodeFactory.AddNodeAsPrototype('Vision/Algebraic Image Operations/F_VN_BitwiseNotImage', node_F_VN_BitwiseNotImage);
NodeFactory.AddNodeAsPrototype('Vision/Algebraic Image Operations/F_VN_BitwiseNotImageExp', node_F_VN_BitwiseNotImageExp);
NodeFactory.AddNodeAsPrototype('Vision/Algebraic Image Operations/F_VN_BitwiseOrImages', node_F_VN_BitwiseOrImages);
NodeFactory.AddNodeAsPrototype('Vision/Algebraic Image Operations/F_VN_BitwiseOrImagesExp', node_F_VN_BitwiseOrImagesExp);
NodeFactory.AddNodeAsPrototype('Vision/Algebraic Image Operations/F_VN_BitwiseOrScalarWithImage', node_F_VN_BitwiseOrScalarWithImage);
NodeFactory.AddNodeAsPrototype('Vision/Algebraic Image Operations/F_VN_BitwiseOrVectorWithImage', node_F_VN_BitwiseOrVectorWithImage);
NodeFactory.AddNodeAsPrototype('Vision/Algebraic Image Operations/F_VN_BitwiseXorImages', node_F_VN_BitwiseXorImages);
NodeFactory.AddNodeAsPrototype('Vision/Algebraic Image Operations/F_VN_BitwiseXorImagesExp', node_F_VN_BitwiseXorImagesExp);
NodeFactory.AddNodeAsPrototype('Vision/Algebraic Image Operations/F_VN_BitwiseXorScalarWithImage', node_F_VN_BitwiseXorScalarWithImage);
NodeFactory.AddNodeAsPrototype('Vision/Algebraic Image Operations/F_VN_BitwiseXorVectorWithImage', node_F_VN_BitwiseXorVectorWithImage);
//NodeFactory.AddNodeAsPrototype('Vision/Algebraic Image Operations/F_VN_BlendImages', node_F_VN_BlendImages);
NodeFactory.AddNodeAsPrototype('Vision/Algebraic Image Operations/F_VN_DivideImageByScalar', node_F_VN_DivideImageByScalar);
NodeFactory.AddNodeAsPrototype('Vision/Algebraic Image Operations/F_VN_DivideImageByVector', node_F_VN_DivideImageByVector);
NodeFactory.AddNodeAsPrototype('Vision/Algebraic Image Operations/F_VN_DivideImages', node_F_VN_DivideImages);
NodeFactory.AddNodeAsPrototype('Vision/Algebraic Image Operations/F_VN_DivideScalarByImage', node_F_VN_DivideScalarByImage);
NodeFactory.AddNodeAsPrototype('Vision/Algebraic Image Operations/F_VN_DivideVectorByImage', node_F_VN_DivideVectorByImage);
NodeFactory.AddNodeAsPrototype('Vision/Algebraic Image Operations/F_VN_ElementwiseExp', node_F_VN_ElementwiseExp);
NodeFactory.AddNodeAsPrototype('Vision/Algebraic Image Operations/F_VN_ElementwiseLog', node_F_VN_ElementwiseLog);
NodeFactory.AddNodeAsPrototype('Vision/Algebraic Image Operations/F_VN_MaxImage', node_F_VN_MaxImage);
NodeFactory.AddNodeAsPrototype('Vision/Algebraic Image Operations/F_VN_MaxImageExp', node_F_VN_MaxImageExp);
NodeFactory.AddNodeAsPrototype('Vision/Algebraic Image Operations/F_VN_MaxImageWithScalar', node_F_VN_MaxImageWithScalar);
NodeFactory.AddNodeAsPrototype('Vision/Algebraic Image Operations/F_VN_MaxImageWithScalarExp', node_F_VN_MaxImageWithScalarExp);
NodeFactory.AddNodeAsPrototype('Vision/Algebraic Image Operations/F_VN_MaxImageWithVector', node_F_VN_MaxImageWithVector);
NodeFactory.AddNodeAsPrototype('Vision/Algebraic Image Operations/F_VN_MaxImageWithVectorExp', node_F_VN_MaxImageWithVectorExp);
NodeFactory.AddNodeAsPrototype('Vision/Algebraic Image Operations/F_VN_MinImage', node_F_VN_MinImage);
NodeFactory.AddNodeAsPrototype('Vision/Algebraic Image Operations/F_VN_MinImageExp', node_F_VN_MinImageExp);
NodeFactory.AddNodeAsPrototype('Vision/Algebraic Image Operations/F_VN_MinImageWithScalar', node_F_VN_MinImageWithScalar);
NodeFactory.AddNodeAsPrototype('Vision/Algebraic Image Operations/F_VN_MinImageWithScalarExp', node_F_VN_MinImageWithScalarExp);
NodeFactory.AddNodeAsPrototype('Vision/Algebraic Image Operations/F_VN_MinImageWithVector', node_F_VN_MinImageWithVector);
NodeFactory.AddNodeAsPrototype('Vision/Algebraic Image Operations/F_VN_MinImageWithVectorExp', node_F_VN_MinImageWithVectorExp);
NodeFactory.AddNodeAsPrototype('Vision/Algebraic Image Operations/F_VN_MultiplyImages', node_F_VN_MultiplyImages);
NodeFactory.AddNodeAsPrototype('Vision/Algebraic Image Operations/F_VN_MultiplyImageWithScalar', node_F_VN_MultiplyImageWithScalar);
NodeFactory.AddNodeAsPrototype('Vision/Algebraic Image Operations/F_VN_MultiplyImageWithVector', node_F_VN_MultiplyImageWithVector);
NodeFactory.AddNodeAsPrototype('Vision/Algebraic Image Operations/F_VN_SubtractImageFromScalar', node_F_VN_SubtractImageFromScalar);
NodeFactory.AddNodeAsPrototype('Vision/Algebraic Image Operations/F_VN_SubtractImageFromVector', node_F_VN_SubtractImageFromVector);
NodeFactory.AddNodeAsPrototype('Vision/Algebraic Image Operations/F_VN_SubtractImages', node_F_VN_SubtractImages);
NodeFactory.AddNodeAsPrototype('Vision/Algebraic Image Operations/F_VN_SubtractScalarFromImage', node_F_VN_SubtractScalarFromImage);
NodeFactory.AddNodeAsPrototype('Vision/Algebraic Image Operations/F_VN_SubtractVectorFromImage', node_F_VN_SubtractVectorFromImage);

// Basic Container Operations
NodeFactory.AddNodeAsPrototype('Vision/Basic Container Operations/F_VN_AppendToContainer/F_VN_AppendToContainer_DINT', node_F_VN_AppendToContainer_DINT);
NodeFactory.AddNodeAsPrototype('Vision/Basic Container Operations/F_VN_AppendToContainer/F_VN_AppendToContainer_INT', node_F_VN_AppendToContainer_INT);
NodeFactory.AddNodeAsPrototype('Vision/Basic Container Operations/F_VN_AppendToContainer/F_VN_AppendToContainer_ITcVnContainer', node_F_VN_AppendToContainer_ITcVnContainer);
//NodeFactory.AddNodeAsPrototype('Vision/Basic Container Operations/F_VN_AppendToContainer/F_VN_AppendToContainer_ITcVnForwardIterator', node_F_VN_AppendToContainer_ITcVnForwardIterator);
NodeFactory.AddNodeAsPrototype('Vision/Basic Container Operations/F_VN_AppendToContainer/F_VN_AppendToContainer_ITcVnImage', node_F_VN_AppendToContainer_ITcVnImage);
NodeFactory.AddNodeAsPrototype('Vision/Basic Container Operations/F_VN_AppendToContainer/F_VN_AppendToContainer_LREAL', node_F_VN_AppendToContainer_LREAL);
NodeFactory.AddNodeAsPrototype('Vision/Basic Container Operations/F_VN_AppendToContainer/F_VN_AppendToContainer_REAL', node_F_VN_AppendToContainer_REAL);
NodeFactory.AddNodeAsPrototype('Vision/Basic Container Operations/F_VN_AppendToContainer/F_VN_AppendToContainer_SINT', node_F_VN_AppendToContainer_SINT);
NodeFactory.AddNodeAsPrototype('Vision/Basic Container Operations/F_VN_AppendToContainer/F_VN_AppendToContainer_TcVnDMatch', node_F_VN_AppendToContainer_TcVnDMatch);
NodeFactory.AddNodeAsPrototype('Vision/Basic Container Operations/F_VN_AppendToContainer/F_VN_AppendToContainer_TcVnKeyPoint', node_F_VN_AppendToContainer_TcVnKeyPoint);
NodeFactory.AddNodeAsPrototype('Vision/Basic Container Operations/F_VN_AppendToContainer/F_VN_AppendToContainer_TcVnPoint2_DINT', node_F_VN_AppendToContainer_TcVnPoint2_DINT);
NodeFactory.AddNodeAsPrototype('Vision/Basic Container Operations/F_VN_AppendToContainer/F_VN_AppendToContainer_TcVnPoint2_LREAL', node_F_VN_AppendToContainer_TcVnPoint2_LREAL);
NodeFactory.AddNodeAsPrototype('Vision/Basic Container Operations/F_VN_AppendToContainer/F_VN_AppendToContainer_TcVnPoint2_REAL', node_F_VN_AppendToContainer_TcVnPoint2_REAL);
NodeFactory.AddNodeAsPrototype('Vision/Basic Container Operations/F_VN_AppendToContainer/F_VN_AppendToContainer_TcVnPoint3_LREAL', node_F_VN_AppendToContainer_TcVnPoint3_LREAL);
NodeFactory.AddNodeAsPrototype('Vision/Basic Container Operations/F_VN_AppendToContainer/F_VN_AppendToContainer_TcVnPoint3_REAL', node_F_VN_AppendToContainer_TcVnPoint3_REAL);
NodeFactory.AddNodeAsPrototype('Vision/Basic Container Operations/F_VN_AppendToContainer/F_VN_AppendToContainer_TcVnRectangle_DINT', node_F_VN_AppendToContainer_TcVnRectangle_DINT);
NodeFactory.AddNodeAsPrototype('Vision/Basic Container Operations/F_VN_AppendToContainer/F_VN_AppendToContainer_TcVnRotatedRectangle', node_F_VN_AppendToContainer_TcVnRotatedRectangle);
NodeFactory.AddNodeAsPrototype('Vision/Basic Container Operations/F_VN_AppendToContainer/F_VN_AppendToContainer_TcVnVector2_DINT', node_F_VN_AppendToContainer_TcVnVector2_DINT);
NodeFactory.AddNodeAsPrototype('Vision/Basic Container Operations/F_VN_AppendToContainer/F_VN_AppendToContainer_TcVnVector2_INT', node_F_VN_AppendToContainer_TcVnVector2_INT);
NodeFactory.AddNodeAsPrototype('Vision/Basic Container Operations/F_VN_AppendToContainer/F_VN_AppendToContainer_TcVnVector2_REAL', node_F_VN_AppendToContainer_TcVnVector2_REAL);
NodeFactory.AddNodeAsPrototype('Vision/Basic Container Operations/F_VN_AppendToContainer/F_VN_AppendToContainer_TcVnVector2_SINT', node_F_VN_AppendToContainer_TcVnVector2_SINT);
NodeFactory.AddNodeAsPrototype('Vision/Basic Container Operations/F_VN_AppendToContainer/F_VN_AppendToContainer_TcVnVector2_UINT', node_F_VN_AppendToContainer_TcVnVector2_UINT);
NodeFactory.AddNodeAsPrototype('Vision/Basic Container Operations/F_VN_AppendToContainer/F_VN_AppendToContainer_TcVnVector2_USINT', node_F_VN_AppendToContainer_TcVnVector2_USINT);
NodeFactory.AddNodeAsPrototype('Vision/Basic Container Operations/F_VN_AppendToContainer/F_VN_AppendToContainer_TcVnVector3_INT', node_F_VN_AppendToContainer_TcVnVector3_INT);
NodeFactory.AddNodeAsPrototype('Vision/Basic Container Operations/F_VN_AppendToContainer/F_VN_AppendToContainer_TcVnVector3_REAL', node_F_VN_AppendToContainer_TcVnVector3_REAL);
NodeFactory.AddNodeAsPrototype('Vision/Basic Container Operations/F_VN_AppendToContainer/F_VN_AppendToContainer_TcVnVector3_SINT', node_F_VN_AppendToContainer_TcVnVector3_SINT);
NodeFactory.AddNodeAsPrototype('Vision/Basic Container Operations/F_VN_AppendToContainer/F_VN_AppendToContainer_TcVnVector3_UINT', node_F_VN_AppendToContainer_TcVnVector3_UINT);
NodeFactory.AddNodeAsPrototype('Vision/Basic Container Operations/F_VN_AppendToContainer/F_VN_AppendToContainer_TcVnVector3_USINT', node_F_VN_AppendToContainer_TcVnVector3_USINT);
NodeFactory.AddNodeAsPrototype('Vision/Basic Container Operations/F_VN_AppendToContainer/F_VN_AppendToContainer_TcVnVector4_DINT', node_F_VN_AppendToContainer_TcVnVector4_DINT);
NodeFactory.AddNodeAsPrototype('Vision/Basic Container Operations/F_VN_AppendToContainer/F_VN_AppendToContainer_TcVnVector4_INT', node_F_VN_AppendToContainer_TcVnVector4_INT);
NodeFactory.AddNodeAsPrototype('Vision/Basic Container Operations/F_VN_AppendToContainer/F_VN_AppendToContainer_TcVnVector4_LREAL', node_F_VN_AppendToContainer_TcVnVector4_LREAL);
NodeFactory.AddNodeAsPrototype('Vision/Basic Container Operations/F_VN_AppendToContainer/F_VN_AppendToContainer_TcVnVector4_REAL', node_F_VN_AppendToContainer_TcVnVector4_REAL);
NodeFactory.AddNodeAsPrototype('Vision/Basic Container Operations/F_VN_AppendToContainer/F_VN_AppendToContainer_TcVnVector4_SINT', node_F_VN_AppendToContainer_TcVnVector4_SINT);
NodeFactory.AddNodeAsPrototype('Vision/Basic Container Operations/F_VN_AppendToContainer/F_VN_AppendToContainer_TcVnVector4_UINT', node_F_VN_AppendToContainer_TcVnVector4_UINT);
NodeFactory.AddNodeAsPrototype('Vision/Basic Container Operations/F_VN_AppendToContainer/F_VN_AppendToContainer_TcVnVector4_USINT', node_F_VN_AppendToContainer_TcVnVector4_USINT);
NodeFactory.AddNodeAsPrototype('Vision/Basic Container Operations/F_VN_AppendToContainer/F_VN_AppendToContainer_UDINT', node_F_VN_AppendToContainer_UDINT);
NodeFactory.AddNodeAsPrototype('Vision/Basic Container Operations/F_VN_AppendToContainer/F_VN_AppendToContainer_UINT', node_F_VN_AppendToContainer_UINT);
NodeFactory.AddNodeAsPrototype('Vision/Basic Container Operations/F_VN_AppendToContainer/F_VN_AppendToContainer_ULINT', node_F_VN_AppendToContainer_ULINT);
NodeFactory.AddNodeAsPrototype('Vision/Basic Container Operations/F_VN_AppendToContainer/F_VN_AppendToContainer_USINT', node_F_VN_AppendToContainer_USINT);

NodeFactory.AddNodeAsPrototype('Vision/Basic Container Operations/F_VN_FillContainer/F_VN_FillContainer_DINT', node_F_VN_FillContainer_DINT);
NodeFactory.AddNodeAsPrototype('Vision/Basic Container Operations/F_VN_FillContainer/F_VN_FillContainer_INT', node_F_VN_FillContainer_INT);
NodeFactory.AddNodeAsPrototype('Vision/Basic Container Operations/F_VN_FillContainer/F_VN_FillContainer_ITcVnImage', node_F_VN_FillContainer_ITcVnImage);
NodeFactory.AddNodeAsPrototype('Vision/Basic Container Operations/F_VN_FillContainer/F_VN_FillContainer_LREAL', node_F_VN_FillContainer_LREAL);
NodeFactory.AddNodeAsPrototype('Vision/Basic Container Operations/F_VN_FillContainer/F_VN_FillContainer_REAL', node_F_VN_FillContainer_REAL);
NodeFactory.AddNodeAsPrototype('Vision/Basic Container Operations/F_VN_FillContainer/F_VN_FillContainer_SINT', node_F_VN_FillContainer_SINT);
NodeFactory.AddNodeAsPrototype('Vision/Basic Container Operations/F_VN_FillContainer/F_VN_FillContainer_TcVnDMatch', node_F_VN_FillContainer_TcVnDMatch);
NodeFactory.AddNodeAsPrototype('Vision/Basic Container Operations/F_VN_FillContainer/F_VN_FillContainer_TcVnKeyPoint', node_F_VN_FillContainer_TcVnKeyPoint);
NodeFactory.AddNodeAsPrototype('Vision/Basic Container Operations/F_VN_FillContainer/F_VN_FillContainer_TcVnPoint2_DINT', node_F_VN_FillContainer_TcVnPoint2_DINT);
NodeFactory.AddNodeAsPrototype('Vision/Basic Container Operations/F_VN_FillContainer/F_VN_FillContainer_TcVnPoint2_LREAL', node_F_VN_FillContainer_TcVnPoint2_LREAL);
NodeFactory.AddNodeAsPrototype('Vision/Basic Container Operations/F_VN_FillContainer/F_VN_FillContainer_TcVnPoint2_REAL', node_F_VN_FillContainer_TcVnPoint2_REAL);
NodeFactory.AddNodeAsPrototype('Vision/Basic Container Operations/F_VN_FillContainer/F_VN_FillContainer_TcVnPoint3_LREAL', node_F_VN_FillContainer_TcVnPoint3_LREAL);
NodeFactory.AddNodeAsPrototype('Vision/Basic Container Operations/F_VN_FillContainer/F_VN_FillContainer_TcVnPoint3_REAL', node_F_VN_FillContainer_TcVnPoint3_REAL);
NodeFactory.AddNodeAsPrototype('Vision/Basic Container Operations/F_VN_FillContainer/F_VN_FillContainer_TcVnRectangle_DINT', node_F_VN_FillContainer_TcVnRectangle_DINT);
NodeFactory.AddNodeAsPrototype('Vision/Basic Container Operations/F_VN_FillContainer/F_VN_FillContainer_TcVnRotatedRectangle', node_F_VN_FillContainer_TcVnRotatedRectangle);
NodeFactory.AddNodeAsPrototype('Vision/Basic Container Operations/F_VN_FillContainer/F_VN_FillContainer_TcVnVector2_DINT', node_F_VN_FillContainer_TcVnVector2_DINT);
NodeFactory.AddNodeAsPrototype('Vision/Basic Container Operations/F_VN_FillContainer/F_VN_FillContainer_TcVnVector2_INT', node_F_VN_FillContainer_TcVnVector2_INT);
NodeFactory.AddNodeAsPrototype('Vision/Basic Container Operations/F_VN_FillContainer/F_VN_FillContainer_TcVnVector2_REAL', node_F_VN_FillContainer_TcVnVector2_REAL);
NodeFactory.AddNodeAsPrototype('Vision/Basic Container Operations/F_VN_FillContainer/F_VN_FillContainer_TcVnVector2_SINT', node_F_VN_FillContainer_TcVnVector2_SINT);
NodeFactory.AddNodeAsPrototype('Vision/Basic Container Operations/F_VN_FillContainer/F_VN_FillContainer_TcVnVector2_UINT', node_F_VN_FillContainer_TcVnVector2_UINT);
NodeFactory.AddNodeAsPrototype('Vision/Basic Container Operations/F_VN_FillContainer/F_VN_FillContainer_TcVnVector2_USINT', node_F_VN_FillContainer_TcVnVector2_USINT);
NodeFactory.AddNodeAsPrototype('Vision/Basic Container Operations/F_VN_FillContainer/F_VN_FillContainer_TcVnVector3_INT', node_F_VN_FillContainer_TcVnVector3_INT);
NodeFactory.AddNodeAsPrototype('Vision/Basic Container Operations/F_VN_FillContainer/F_VN_FillContainer_TcVnVector3_REAL', node_F_VN_FillContainer_TcVnVector3_REAL);
NodeFactory.AddNodeAsPrototype('Vision/Basic Container Operations/F_VN_FillContainer/F_VN_FillContainer_TcVnVector3_SINT', node_F_VN_FillContainer_TcVnVector3_SINT);
NodeFactory.AddNodeAsPrototype('Vision/Basic Container Operations/F_VN_FillContainer/F_VN_FillContainer_TcVnVector3_UINT', node_F_VN_FillContainer_TcVnVector3_UINT);
NodeFactory.AddNodeAsPrototype('Vision/Basic Container Operations/F_VN_FillContainer/F_VN_FillContainer_TcVnVector3_USINT', node_F_VN_FillContainer_TcVnVector3_USINT);
NodeFactory.AddNodeAsPrototype('Vision/Basic Container Operations/F_VN_FillContainer/F_VN_FillContainer_TcVnVector4_DINT', node_F_VN_FillContainer_TcVnVector4_DINT);
NodeFactory.AddNodeAsPrototype('Vision/Basic Container Operations/F_VN_FillContainer/F_VN_FillContainer_TcVnVector4_INT', node_F_VN_FillContainer_TcVnVector4_INT);
NodeFactory.AddNodeAsPrototype('Vision/Basic Container Operations/F_VN_FillContainer/F_VN_FillContainer_TcVnVector4_LREAL', node_F_VN_FillContainer_TcVnVector4_LREAL);
NodeFactory.AddNodeAsPrototype('Vision/Basic Container Operations/F_VN_FillContainer/F_VN_FillContainer_TcVnVector4_REAL', node_F_VN_FillContainer_TcVnVector4_REAL);
NodeFactory.AddNodeAsPrototype('Vision/Basic Container Operations/F_VN_FillContainer/F_VN_FillContainer_TcVnVector4_SINT', node_F_VN_FillContainer_TcVnVector4_SINT);
NodeFactory.AddNodeAsPrototype('Vision/Basic Container Operations/F_VN_FillContainer/F_VN_FillContainer_TcVnVector4_UINT', node_F_VN_FillContainer_TcVnVector4_UINT);
NodeFactory.AddNodeAsPrototype('Vision/Basic Container Operations/F_VN_FillContainer/F_VN_FillContainer_TcVnVector4_USINT', node_F_VN_FillContainer_TcVnVector4_USINT);
NodeFactory.AddNodeAsPrototype('Vision/Basic Container Operations/F_VN_FillContainer/F_VN_FillContainer_UDINT', node_F_VN_FillContainer_UDINT);
NodeFactory.AddNodeAsPrototype('Vision/Basic Container Operations/F_VN_FillContainer/F_VN_FillContainer_UINT', node_F_VN_FillContainer_UINT);
NodeFactory.AddNodeAsPrototype('Vision/Basic Container Operations/F_VN_FillContainer/F_VN_FillContainer_ULINT', node_F_VN_FillContainer_ULINT);
NodeFactory.AddNodeAsPrototype('Vision/Basic Container Operations/F_VN_FillContainer/F_VN_FillContainer_USINT', node_F_VN_FillContainer_USINT);

NodeFactory.AddNodeAsPrototype('Vision/Basic Container Operations/F_VN_FillContainerExp/F_VN_FillContainerExp_DINT', node_F_VN_FillContainerExp_DINT);
NodeFactory.AddNodeAsPrototype('Vision/Basic Container Operations/F_VN_FillContainerExp/F_VN_FillContainerExp_INT', node_F_VN_FillContainerExp_INT);
NodeFactory.AddNodeAsPrototype('Vision/Basic Container Operations/F_VN_FillContainerExp/F_VN_FillContainerExp_ITcVnImage', node_F_VN_FillContainerExp_ITcVnImage);
NodeFactory.AddNodeAsPrototype('Vision/Basic Container Operations/F_VN_FillContainerExp/F_VN_FillContainerExp_LREAL', node_F_VN_FillContainerExp_LREAL);
NodeFactory.AddNodeAsPrototype('Vision/Basic Container Operations/F_VN_FillContainerExp/F_VN_FillContainerExp_REAL', node_F_VN_FillContainerExp_REAL);
NodeFactory.AddNodeAsPrototype('Vision/Basic Container Operations/F_VN_FillContainerExp/F_VN_FillContainerExp_SINT', node_F_VN_FillContainerExp_SINT);
NodeFactory.AddNodeAsPrototype('Vision/Basic Container Operations/F_VN_FillContainerExp/F_VN_FillContainerExp_TcVnDMatch', node_F_VN_FillContainerExp_TcVnDMatch);
NodeFactory.AddNodeAsPrototype('Vision/Basic Container Operations/F_VN_FillContainerExp/F_VN_FillContainerExp_TcVnKeyPoint', node_F_VN_FillContainerExp_TcVnKeyPoint);
NodeFactory.AddNodeAsPrototype('Vision/Basic Container Operations/F_VN_FillContainerExp/F_VN_FillContainerExp_TcVnPoint2_DINT', node_F_VN_FillContainerExp_TcVnPoint2_DINT);
NodeFactory.AddNodeAsPrototype('Vision/Basic Container Operations/F_VN_FillContainerExp/F_VN_FillContainerExp_TcVnPoint2_LREAL', node_F_VN_FillContainerExp_TcVnPoint2_LREAL);
NodeFactory.AddNodeAsPrototype('Vision/Basic Container Operations/F_VN_FillContainerExp/F_VN_FillContainerExp_TcVnPoint2_REAL', node_F_VN_FillContainerExp_TcVnPoint2_REAL);
NodeFactory.AddNodeAsPrototype('Vision/Basic Container Operations/F_VN_FillContainerExp/F_VN_FillContainerExp_TcVnPoint3_LREAL', node_F_VN_FillContainerExp_TcVnPoint3_LREAL);
NodeFactory.AddNodeAsPrototype('Vision/Basic Container Operations/F_VN_FillContainerExp/F_VN_FillContainerExp_TcVnPoint3_REAL', node_F_VN_FillContainerExp_TcVnPoint3_REAL);
NodeFactory.AddNodeAsPrototype('Vision/Basic Container Operations/F_VN_FillContainerExp/F_VN_FillContainerExp_TcVnRectangle_DINT', node_F_VN_FillContainerExp_TcVnRectangle_DINT);
NodeFactory.AddNodeAsPrototype('Vision/Basic Container Operations/F_VN_FillContainerExp/F_VN_FillContainerExp_TcVnRotatedRectangle', node_F_VN_FillContainerExp_TcVnRotatedRectangle);
NodeFactory.AddNodeAsPrototype('Vision/Basic Container Operations/F_VN_FillContainerExp/F_VN_FillContainerExp_TcVnVector2_DINT', node_F_VN_FillContainerExp_TcVnVector2_DINT);
NodeFactory.AddNodeAsPrototype('Vision/Basic Container Operations/F_VN_FillContainerExp/F_VN_FillContainerExp_TcVnVector2_INT', node_F_VN_FillContainerExp_TcVnVector2_INT);
NodeFactory.AddNodeAsPrototype('Vision/Basic Container Operations/F_VN_FillContainerExp/F_VN_FillContainerExp_TcVnVector2_REAL', node_F_VN_FillContainerExp_TcVnVector2_REAL);
NodeFactory.AddNodeAsPrototype('Vision/Basic Container Operations/F_VN_FillContainerExp/F_VN_FillContainerExp_TcVnVector2_SINT', node_F_VN_FillContainerExp_TcVnVector2_SINT);
NodeFactory.AddNodeAsPrototype('Vision/Basic Container Operations/F_VN_FillContainerExp/F_VN_FillContainerExp_TcVnVector2_UINT', node_F_VN_FillContainerExp_TcVnVector2_UINT);
NodeFactory.AddNodeAsPrototype('Vision/Basic Container Operations/F_VN_FillContainerExp/F_VN_FillContainerExp_TcVnVector2_USINT', node_F_VN_FillContainerExp_TcVnVector2_USINT);
NodeFactory.AddNodeAsPrototype('Vision/Basic Container Operations/F_VN_FillContainerExp/F_VN_FillContainerExp_TcVnVector3_INT', node_F_VN_FillContainerExp_TcVnVector3_INT);
NodeFactory.AddNodeAsPrototype('Vision/Basic Container Operations/F_VN_FillContainerExp/F_VN_FillContainerExp_TcVnVector3_REAL', node_F_VN_FillContainerExp_TcVnVector3_REAL);
NodeFactory.AddNodeAsPrototype('Vision/Basic Container Operations/F_VN_FillContainerExp/F_VN_FillContainerExp_TcVnVector3_SINT', node_F_VN_FillContainerExp_TcVnVector3_SINT);
NodeFactory.AddNodeAsPrototype('Vision/Basic Container Operations/F_VN_FillContainerExp/F_VN_FillContainerExp_TcVnVector3_UINT', node_F_VN_FillContainerExp_TcVnVector3_UINT);
NodeFactory.AddNodeAsPrototype('Vision/Basic Container Operations/F_VN_FillContainerExp/F_VN_FillContainerExp_TcVnVector3_USINT', node_F_VN_FillContainerExp_TcVnVector3_USINT);
NodeFactory.AddNodeAsPrototype('Vision/Basic Container Operations/F_VN_FillContainerExp/F_VN_FillContainerExp_TcVnVector4_DINT', node_F_VN_FillContainerExp_TcVnVector4_DINT);
NodeFactory.AddNodeAsPrototype('Vision/Basic Container Operations/F_VN_FillContainerExp/F_VN_FillContainerExp_TcVnVector4_INT', node_F_VN_FillContainerExp_TcVnVector4_INT);
NodeFactory.AddNodeAsPrototype('Vision/Basic Container Operations/F_VN_FillContainerExp/F_VN_FillContainerExp_TcVnVector4_LREAL', node_F_VN_FillContainerExp_TcVnVector4_LREAL);
NodeFactory.AddNodeAsPrototype('Vision/Basic Container Operations/F_VN_FillContainerExp/F_VN_FillContainerExp_TcVnVector4_REAL', node_F_VN_FillContainerExp_TcVnVector4_REAL);
NodeFactory.AddNodeAsPrototype('Vision/Basic Container Operations/F_VN_FillContainerExp/F_VN_FillContainerExp_TcVnVector4_SINT', node_F_VN_FillContainerExp_TcVnVector4_SINT);
NodeFactory.AddNodeAsPrototype('Vision/Basic Container Operations/F_VN_FillContainerExp/F_VN_FillContainerExp_TcVnVector4_UINT', node_F_VN_FillContainerExp_TcVnVector4_UINT);
NodeFactory.AddNodeAsPrototype('Vision/Basic Container Operations/F_VN_FillContainerExp/F_VN_FillContainerExp_TcVnVector4_USINT', node_F_VN_FillContainerExp_TcVnVector4_USINT);
NodeFactory.AddNodeAsPrototype('Vision/Basic Container Operations/F_VN_FillContainerExp/F_VN_FillContainerExp_UDINT', node_F_VN_FillContainerExp_UDINT);
NodeFactory.AddNodeAsPrototype('Vision/Basic Container Operations/F_VN_FillContainerExp/F_VN_FillContainerExp_UINT', node_F_VN_FillContainerExp_UINT);
NodeFactory.AddNodeAsPrototype('Vision/Basic Container Operations/F_VN_FillContainerExp/F_VN_FillContainerExp_ULINT', node_F_VN_FillContainerExp_ULINT);
NodeFactory.AddNodeAsPrototype('Vision/Basic Container Operations/F_VN_FillContainerExp/F_VN_FillContainerExp_USINT', node_F_VN_FillContainerExp_USINT);

NodeFactory.AddNodeAsPrototype('Vision/Basic Container Operations/F_VN_GetAt/F_VN_GetAt_DINT', node_F_VN_GetAt_DINT);
NodeFactory.AddNodeAsPrototype('Vision/Basic Container Operations/F_VN_GetAt/F_VN_GetAt_INT', node_F_VN_GetAt_INT);
NodeFactory.AddNodeAsPrototype('Vision/Basic Container Operations/F_VN_GetAt/F_VN_GetAt_ITcVnContainer', node_F_VN_GetAt_ITcVnContainer);
NodeFactory.AddNodeAsPrototype('Vision/Basic Container Operations/F_VN_GetAt/F_VN_GetAt_ITcVnImage', node_F_VN_GetAt_ITcVnImage);
NodeFactory.AddNodeAsPrototype('Vision/Basic Container Operations/F_VN_GetAt/F_VN_GetAt_LREAL', node_F_VN_GetAt_LREAL);
NodeFactory.AddNodeAsPrototype('Vision/Basic Container Operations/F_VN_GetAt/F_VN_GetAt_REAL', node_F_VN_GetAt_REAL);
NodeFactory.AddNodeAsPrototype('Vision/Basic Container Operations/F_VN_GetAt/F_VN_GetAt_SINT', node_F_VN_GetAt_SINT);
NodeFactory.AddNodeAsPrototype('Vision/Basic Container Operations/F_VN_GetAt/F_VN_GetAt_TcVnDMatch', node_F_VN_GetAt_TcVnDMatch);
NodeFactory.AddNodeAsPrototype('Vision/Basic Container Operations/F_VN_GetAt/F_VN_GetAt_TcVnKeyPoint', node_F_VN_GetAt_TcVnKeyPoint);
NodeFactory.AddNodeAsPrototype('Vision/Basic Container Operations/F_VN_GetAt/F_VN_GetAt_TcVnPoint2_DINT', node_F_VN_GetAt_TcVnPoint2_DINT);
NodeFactory.AddNodeAsPrototype('Vision/Basic Container Operations/F_VN_GetAt/F_VN_GetAt_TcVnPoint2_LREAL', node_F_VN_GetAt_TcVnPoint2_LREAL);
NodeFactory.AddNodeAsPrototype('Vision/Basic Container Operations/F_VN_GetAt/F_VN_GetAt_TcVnPoint2_REAL', node_F_VN_GetAt_TcVnPoint2_REAL);
NodeFactory.AddNodeAsPrototype('Vision/Basic Container Operations/F_VN_GetAt/F_VN_GetAt_TcVnPoint3_LREAL', node_F_VN_GetAt_TcVnPoint3_LREAL);
NodeFactory.AddNodeAsPrototype('Vision/Basic Container Operations/F_VN_GetAt/F_VN_GetAt_TcVnPoint3_REAL', node_F_VN_GetAt_TcVnPoint3_REAL);
NodeFactory.AddNodeAsPrototype('Vision/Basic Container Operations/F_VN_GetAt/F_VN_GetAt_TcVnRectangle_DINT', node_F_VN_GetAt_TcVnRectangle_DINT);
NodeFactory.AddNodeAsPrototype('Vision/Basic Container Operations/F_VN_GetAt/F_VN_GetAt_TcVnRotatedRectangle', node_F_VN_GetAt_TcVnRotatedRectangle);
NodeFactory.AddNodeAsPrototype('Vision/Basic Container Operations/F_VN_GetAt/F_VN_GetAt_TcVnVector2_DINT', node_F_VN_GetAt_TcVnVector2_DINT);
NodeFactory.AddNodeAsPrototype('Vision/Basic Container Operations/F_VN_GetAt/F_VN_GetAt_TcVnVector2_INT', node_F_VN_GetAt_TcVnVector2_INT);
NodeFactory.AddNodeAsPrototype('Vision/Basic Container Operations/F_VN_GetAt/F_VN_GetAt_TcVnVector2_REAL', node_F_VN_GetAt_TcVnVector2_REAL);
NodeFactory.AddNodeAsPrototype('Vision/Basic Container Operations/F_VN_GetAt/F_VN_GetAt_TcVnVector2_SINT', node_F_VN_GetAt_TcVnVector2_SINT);
NodeFactory.AddNodeAsPrototype('Vision/Basic Container Operations/F_VN_GetAt/F_VN_GetAt_TcVnVector2_UINT', node_F_VN_GetAt_TcVnVector2_UINT);
NodeFactory.AddNodeAsPrototype('Vision/Basic Container Operations/F_VN_GetAt/F_VN_GetAt_TcVnVector2_USINT', node_F_VN_GetAt_TcVnVector2_USINT);
NodeFactory.AddNodeAsPrototype('Vision/Basic Container Operations/F_VN_GetAt/F_VN_GetAt_TcVnVector3_INT', node_F_VN_GetAt_TcVnVector3_INT);
NodeFactory.AddNodeAsPrototype('Vision/Basic Container Operations/F_VN_GetAt/F_VN_GetAt_TcVnVector3_REAL', node_F_VN_GetAt_TcVnVector3_REAL);
NodeFactory.AddNodeAsPrototype('Vision/Basic Container Operations/F_VN_GetAt/F_VN_GetAt_TcVnVector3_SINT', node_F_VN_GetAt_TcVnVector3_SINT);
NodeFactory.AddNodeAsPrototype('Vision/Basic Container Operations/F_VN_GetAt/F_VN_GetAt_TcVnVector3_UINT', node_F_VN_GetAt_TcVnVector3_UINT);
NodeFactory.AddNodeAsPrototype('Vision/Basic Container Operations/F_VN_GetAt/F_VN_GetAt_TcVnVector3_USINT', node_F_VN_GetAt_TcVnVector3_USINT);
NodeFactory.AddNodeAsPrototype('Vision/Basic Container Operations/F_VN_GetAt/F_VN_GetAt_TcVnVector4_DINT', node_F_VN_GetAt_TcVnVector4_DINT);
NodeFactory.AddNodeAsPrototype('Vision/Basic Container Operations/F_VN_GetAt/F_VN_GetAt_TcVnVector4_INT', node_F_VN_GetAt_TcVnVector4_INT);
NodeFactory.AddNodeAsPrototype('Vision/Basic Container Operations/F_VN_GetAt/F_VN_GetAt_TcVnVector4_LREAL', node_F_VN_GetAt_TcVnVector4_LREAL);
NodeFactory.AddNodeAsPrototype('Vision/Basic Container Operations/F_VN_GetAt/F_VN_GetAt_TcVnVector4_REAL', node_F_VN_GetAt_TcVnVector4_REAL);
NodeFactory.AddNodeAsPrototype('Vision/Basic Container Operations/F_VN_GetAt/F_VN_GetAt_TcVnVector4_SINT', node_F_VN_GetAt_TcVnVector4_SINT);
NodeFactory.AddNodeAsPrototype('Vision/Basic Container Operations/F_VN_GetAt/F_VN_GetAt_TcVnVector4_UINT', node_F_VN_GetAt_TcVnVector4_UINT);
NodeFactory.AddNodeAsPrototype('Vision/Basic Container Operations/F_VN_GetAt/F_VN_GetAt_TcVnVector4_USINT', node_F_VN_GetAt_TcVnVector4_USINT);
NodeFactory.AddNodeAsPrototype('Vision/Basic Container Operations/F_VN_GetAt/F_VN_GetAt_UDINT', node_F_VN_GetAt_UDINT);
NodeFactory.AddNodeAsPrototype('Vision/Basic Container Operations/F_VN_GetAt/F_VN_GetAt_UINT', node_F_VN_GetAt_UINT);
NodeFactory.AddNodeAsPrototype('Vision/Basic Container Operations/F_VN_GetAt/F_VN_GetAt_ULINT', node_F_VN_GetAt_ULINT);
NodeFactory.AddNodeAsPrototype('Vision/Basic Container Operations/F_VN_GetAt/F_VN_GetAt_USINT', node_F_VN_GetAt_USINT);

NodeFactory.AddNodeAsPrototype('Vision/Basic Container Operations/F_VN_InsertIntoContainer/F_VN_InsertIntoContainer_DINT', node_F_VN_InsertIntoContainer_DINT);
NodeFactory.AddNodeAsPrototype('Vision/Basic Container Operations/F_VN_InsertIntoContainer/F_VN_InsertIntoContainer_INT', node_F_VN_InsertIntoContainer_INT);
NodeFactory.AddNodeAsPrototype('Vision/Basic Container Operations/F_VN_InsertIntoContainer/F_VN_InsertIntoContainer_ITcVnContainer', node_F_VN_InsertIntoContainer_ITcVnContainer);
//NodeFactory.AddNodeAsPrototype('Vision/Basic Container Operations/F_VN_InsertIntoContainer/F_VN_InsertIntoContainer_ITcVnForwardIterator', node_F_VN_InsertIntoContainer_ITcVnForwardIterator);
NodeFactory.AddNodeAsPrototype('Vision/Basic Container Operations/F_VN_InsertIntoContainer/F_VN_InsertIntoContainer_ITcVnImage', node_F_VN_InsertIntoContainer_ITcVnImage);
NodeFactory.AddNodeAsPrototype('Vision/Basic Container Operations/F_VN_InsertIntoContainer/F_VN_InsertIntoContainer_LREAL', node_F_VN_InsertIntoContainer_LREAL);
NodeFactory.AddNodeAsPrototype('Vision/Basic Container Operations/F_VN_InsertIntoContainer/F_VN_InsertIntoContainer_REAL', node_F_VN_InsertIntoContainer_REAL);
NodeFactory.AddNodeAsPrototype('Vision/Basic Container Operations/F_VN_InsertIntoContainer/F_VN_InsertIntoContainer_SINT', node_F_VN_InsertIntoContainer_SINT);
NodeFactory.AddNodeAsPrototype('Vision/Basic Container Operations/F_VN_InsertIntoContainer/F_VN_InsertIntoContainer_TcVnDMatch', node_F_VN_InsertIntoContainer_TcVnDMatch);
NodeFactory.AddNodeAsPrototype('Vision/Basic Container Operations/F_VN_InsertIntoContainer/F_VN_InsertIntoContainer_TcVnKeyPoint', node_F_VN_InsertIntoContainer_TcVnKeyPoint);
NodeFactory.AddNodeAsPrototype('Vision/Basic Container Operations/F_VN_InsertIntoContainer/F_VN_InsertIntoContainer_TcVnPoint2_DINT', node_F_VN_InsertIntoContainer_TcVnPoint2_DINT);
NodeFactory.AddNodeAsPrototype('Vision/Basic Container Operations/F_VN_InsertIntoContainer/F_VN_InsertIntoContainer_TcVnPoint2_LREAL', node_F_VN_InsertIntoContainer_TcVnPoint2_LREAL);
NodeFactory.AddNodeAsPrototype('Vision/Basic Container Operations/F_VN_InsertIntoContainer/F_VN_InsertIntoContainer_TcVnPoint2_REAL', node_F_VN_InsertIntoContainer_TcVnPoint2_REAL);
NodeFactory.AddNodeAsPrototype('Vision/Basic Container Operations/F_VN_InsertIntoContainer/F_VN_InsertIntoContainer_TcVnPoint3_LREAL', node_F_VN_InsertIntoContainer_TcVnPoint3_LREAL);
NodeFactory.AddNodeAsPrototype('Vision/Basic Container Operations/F_VN_InsertIntoContainer/F_VN_InsertIntoContainer_TcVnPoint3_REAL', node_F_VN_InsertIntoContainer_TcVnPoint3_REAL);
NodeFactory.AddNodeAsPrototype('Vision/Basic Container Operations/F_VN_InsertIntoContainer/F_VN_InsertIntoContainer_TcVnRectangle_DINT', node_F_VN_InsertIntoContainer_TcVnRectangle_DINT);
NodeFactory.AddNodeAsPrototype('Vision/Basic Container Operations/F_VN_InsertIntoContainer/F_VN_InsertIntoContainer_TcVnRotatedRectangle', node_F_VN_InsertIntoContainer_TcVnRotatedRectangle);
NodeFactory.AddNodeAsPrototype('Vision/Basic Container Operations/F_VN_InsertIntoContainer/F_VN_InsertIntoContainer_TcVnVector2_DINT', node_F_VN_InsertIntoContainer_TcVnVector2_DINT);
NodeFactory.AddNodeAsPrototype('Vision/Basic Container Operations/F_VN_InsertIntoContainer/F_VN_InsertIntoContainer_TcVnVector2_INT', node_F_VN_InsertIntoContainer_TcVnVector2_INT);
NodeFactory.AddNodeAsPrototype('Vision/Basic Container Operations/F_VN_InsertIntoContainer/F_VN_InsertIntoContainer_TcVnVector2_REAL', node_F_VN_InsertIntoContainer_TcVnVector2_REAL);
NodeFactory.AddNodeAsPrototype('Vision/Basic Container Operations/F_VN_InsertIntoContainer/F_VN_InsertIntoContainer_TcVnVector2_SINT', node_F_VN_InsertIntoContainer_TcVnVector2_SINT);
NodeFactory.AddNodeAsPrototype('Vision/Basic Container Operations/F_VN_InsertIntoContainer/F_VN_InsertIntoContainer_TcVnVector2_UINT', node_F_VN_InsertIntoContainer_TcVnVector2_UINT);
NodeFactory.AddNodeAsPrototype('Vision/Basic Container Operations/F_VN_InsertIntoContainer/F_VN_InsertIntoContainer_TcVnVector2_USINT', node_F_VN_InsertIntoContainer_TcVnVector2_USINT);
NodeFactory.AddNodeAsPrototype('Vision/Basic Container Operations/F_VN_InsertIntoContainer/F_VN_InsertIntoContainer_TcVnVector3_INT', node_F_VN_InsertIntoContainer_TcVnVector3_INT);
NodeFactory.AddNodeAsPrototype('Vision/Basic Container Operations/F_VN_InsertIntoContainer/F_VN_InsertIntoContainer_TcVnVector3_REAL', node_F_VN_InsertIntoContainer_TcVnVector3_REAL);
NodeFactory.AddNodeAsPrototype('Vision/Basic Container Operations/F_VN_InsertIntoContainer/F_VN_InsertIntoContainer_TcVnVector3_SINT', node_F_VN_InsertIntoContainer_TcVnVector3_SINT);
NodeFactory.AddNodeAsPrototype('Vision/Basic Container Operations/F_VN_InsertIntoContainer/F_VN_InsertIntoContainer_TcVnVector3_UINT', node_F_VN_InsertIntoContainer_TcVnVector3_UINT);
NodeFactory.AddNodeAsPrototype('Vision/Basic Container Operations/F_VN_InsertIntoContainer/F_VN_InsertIntoContainer_TcVnVector3_USINT', node_F_VN_InsertIntoContainer_TcVnVector3_USINT);
NodeFactory.AddNodeAsPrototype('Vision/Basic Container Operations/F_VN_InsertIntoContainer/F_VN_InsertIntoContainer_TcVnVector4_DINT', node_F_VN_InsertIntoContainer_TcVnVector4_DINT);
NodeFactory.AddNodeAsPrototype('Vision/Basic Container Operations/F_VN_InsertIntoContainer/F_VN_InsertIntoContainer_TcVnVector4_INT', node_F_VN_InsertIntoContainer_TcVnVector4_INT);
NodeFactory.AddNodeAsPrototype('Vision/Basic Container Operations/F_VN_InsertIntoContainer/F_VN_InsertIntoContainer_TcVnVector4_LREAL', node_F_VN_InsertIntoContainer_TcVnVector4_LREAL);
NodeFactory.AddNodeAsPrototype('Vision/Basic Container Operations/F_VN_InsertIntoContainer/F_VN_InsertIntoContainer_TcVnVector4_REAL', node_F_VN_InsertIntoContainer_TcVnVector4_REAL);
NodeFactory.AddNodeAsPrototype('Vision/Basic Container Operations/F_VN_InsertIntoContainer/F_VN_InsertIntoContainer_TcVnVector4_SINT', node_F_VN_InsertIntoContainer_TcVnVector4_SINT);
NodeFactory.AddNodeAsPrototype('Vision/Basic Container Operations/F_VN_InsertIntoContainer/F_VN_InsertIntoContainer_TcVnVector4_UINT', node_F_VN_InsertIntoContainer_TcVnVector4_UINT);
NodeFactory.AddNodeAsPrototype('Vision/Basic Container Operations/F_VN_InsertIntoContainer/F_VN_InsertIntoContainer_TcVnVector4_USINT', node_F_VN_InsertIntoContainer_TcVnVector4_USINT);
NodeFactory.AddNodeAsPrototype('Vision/Basic Container Operations/F_VN_InsertIntoContainer/F_VN_InsertIntoContainer_UDINT', node_F_VN_InsertIntoContainer_UDINT);
NodeFactory.AddNodeAsPrototype('Vision/Basic Container Operations/F_VN_InsertIntoContainer/F_VN_InsertIntoContainer_UINT', node_F_VN_InsertIntoContainer_UINT);
NodeFactory.AddNodeAsPrototype('Vision/Basic Container Operations/F_VN_InsertIntoContainer/F_VN_InsertIntoContainer_ULINT', node_F_VN_InsertIntoContainer_ULINT);
NodeFactory.AddNodeAsPrototype('Vision/Basic Container Operations/F_VN_InsertIntoContainer/F_VN_InsertIntoContainer_USINT', node_F_VN_InsertIntoContainer_USINT);

NodeFactory.AddNodeAsPrototype('Vision/Basic Container Operations/F_VN_SetAt/F_VN_SetAt_DINT', node_F_VN_SetAt_DINT);
NodeFactory.AddNodeAsPrototype('Vision/Basic Container Operations/F_VN_SetAt/F_VN_SetAt_INT', node_F_VN_SetAt_INT);
NodeFactory.AddNodeAsPrototype('Vision/Basic Container Operations/F_VN_SetAt/F_VN_SetAt_ITcVnContainer', node_F_VN_SetAt_ITcVnContainer);
NodeFactory.AddNodeAsPrototype('Vision/Basic Container Operations/F_VN_SetAt/F_VN_SetAt_ITcVnImage', node_F_VN_SetAt_ITcVnImage);
NodeFactory.AddNodeAsPrototype('Vision/Basic Container Operations/F_VN_SetAt/F_VN_SetAt_LREAL', node_F_VN_SetAt_LREAL);
NodeFactory.AddNodeAsPrototype('Vision/Basic Container Operations/F_VN_SetAt/F_VN_SetAt_REAL', node_F_VN_SetAt_REAL);
NodeFactory.AddNodeAsPrototype('Vision/Basic Container Operations/F_VN_SetAt/F_VN_SetAt_SINT', node_F_VN_SetAt_SINT);
NodeFactory.AddNodeAsPrototype('Vision/Basic Container Operations/F_VN_SetAt/F_VN_SetAt_TcVnDMatch', node_F_VN_SetAt_TcVnDMatch);
NodeFactory.AddNodeAsPrototype('Vision/Basic Container Operations/F_VN_SetAt/F_VN_SetAt_TcVnKeyPoint', node_F_VN_SetAt_TcVnKeyPoint);
NodeFactory.AddNodeAsPrototype('Vision/Basic Container Operations/F_VN_SetAt/F_VN_SetAt_TcVnPoint2_DINT', node_F_VN_SetAt_TcVnPoint2_DINT);
NodeFactory.AddNodeAsPrototype('Vision/Basic Container Operations/F_VN_SetAt/F_VN_SetAt_TcVnPoint2_LREAL', node_F_VN_SetAt_TcVnPoint2_LREAL);
NodeFactory.AddNodeAsPrototype('Vision/Basic Container Operations/F_VN_SetAt/F_VN_SetAt_TcVnPoint2_REAL', node_F_VN_SetAt_TcVnPoint2_REAL);
NodeFactory.AddNodeAsPrototype('Vision/Basic Container Operations/F_VN_SetAt/F_VN_SetAt_TcVnPoint3_LREAL', node_F_VN_SetAt_TcVnPoint3_LREAL);
NodeFactory.AddNodeAsPrototype('Vision/Basic Container Operations/F_VN_SetAt/F_VN_SetAt_TcVnPoint3_REAL', node_F_VN_SetAt_TcVnPoint3_REAL);
NodeFactory.AddNodeAsPrototype('Vision/Basic Container Operations/F_VN_SetAt/F_VN_SetAt_TcVnRectangle_DINT', node_F_VN_SetAt_TcVnRectangle_DINT);
NodeFactory.AddNodeAsPrototype('Vision/Basic Container Operations/F_VN_SetAt/F_VN_SetAt_TcVnRotatedRectangle', node_F_VN_SetAt_TcVnRotatedRectangle);
NodeFactory.AddNodeAsPrototype('Vision/Basic Container Operations/F_VN_SetAt/F_VN_SetAt_TcVnVector2_DINT', node_F_VN_SetAt_TcVnVector2_DINT);
NodeFactory.AddNodeAsPrototype('Vision/Basic Container Operations/F_VN_SetAt/F_VN_SetAt_TcVnVector2_INT', node_F_VN_SetAt_TcVnVector2_INT);
NodeFactory.AddNodeAsPrototype('Vision/Basic Container Operations/F_VN_SetAt/F_VN_SetAt_TcVnVector2_REAL', node_F_VN_SetAt_TcVnVector2_REAL);
NodeFactory.AddNodeAsPrototype('Vision/Basic Container Operations/F_VN_SetAt/F_VN_SetAt_TcVnVector2_SINT', node_F_VN_SetAt_TcVnVector2_SINT);
NodeFactory.AddNodeAsPrototype('Vision/Basic Container Operations/F_VN_SetAt/F_VN_SetAt_TcVnVector2_UINT', node_F_VN_SetAt_TcVnVector2_UINT);
NodeFactory.AddNodeAsPrototype('Vision/Basic Container Operations/F_VN_SetAt/F_VN_SetAt_TcVnVector2_USINT', node_F_VN_SetAt_TcVnVector2_USINT);
NodeFactory.AddNodeAsPrototype('Vision/Basic Container Operations/F_VN_SetAt/F_VN_SetAt_TcVnVector3_INT', node_F_VN_SetAt_TcVnVector3_INT);
NodeFactory.AddNodeAsPrototype('Vision/Basic Container Operations/F_VN_SetAt/F_VN_SetAt_TcVnVector3_REAL', node_F_VN_SetAt_TcVnVector3_REAL);
NodeFactory.AddNodeAsPrototype('Vision/Basic Container Operations/F_VN_SetAt/F_VN_SetAt_TcVnVector3_SINT', node_F_VN_SetAt_TcVnVector3_SINT);
NodeFactory.AddNodeAsPrototype('Vision/Basic Container Operations/F_VN_SetAt/F_VN_SetAt_TcVnVector3_UINT', node_F_VN_SetAt_TcVnVector3_UINT);
NodeFactory.AddNodeAsPrototype('Vision/Basic Container Operations/F_VN_SetAt/F_VN_SetAt_TcVnVector3_USINT', node_F_VN_SetAt_TcVnVector3_USINT);
NodeFactory.AddNodeAsPrototype('Vision/Basic Container Operations/F_VN_SetAt/F_VN_SetAt_TcVnVector4_DINT', node_F_VN_SetAt_TcVnVector4_DINT);
NodeFactory.AddNodeAsPrototype('Vision/Basic Container Operations/F_VN_SetAt/F_VN_SetAt_TcVnVector4_INT', node_F_VN_SetAt_TcVnVector4_INT);
NodeFactory.AddNodeAsPrototype('Vision/Basic Container Operations/F_VN_SetAt/F_VN_SetAt_TcVnVector4_LREAL', node_F_VN_SetAt_TcVnVector4_LREAL);
NodeFactory.AddNodeAsPrototype('Vision/Basic Container Operations/F_VN_SetAt/F_VN_SetAt_TcVnVector4_REAL', node_F_VN_SetAt_TcVnVector4_REAL);
NodeFactory.AddNodeAsPrototype('Vision/Basic Container Operations/F_VN_SetAt/F_VN_SetAt_TcVnVector4_SINT', node_F_VN_SetAt_TcVnVector4_SINT);
NodeFactory.AddNodeAsPrototype('Vision/Basic Container Operations/F_VN_SetAt/F_VN_SetAt_TcVnVector4_UINT', node_F_VN_SetAt_TcVnVector4_UINT);
NodeFactory.AddNodeAsPrototype('Vision/Basic Container Operations/F_VN_SetAt/F_VN_SetAt_TcVnVector4_USINT', node_F_VN_SetAt_TcVnVector4_USINT);
NodeFactory.AddNodeAsPrototype('Vision/Basic Container Operations/F_VN_SetAt/F_VN_SetAt_UDINT', node_F_VN_SetAt_UDINT);
NodeFactory.AddNodeAsPrototype('Vision/Basic Container Operations/F_VN_SetAt/F_VN_SetAt_UINT', node_F_VN_SetAt_UINT);
NodeFactory.AddNodeAsPrototype('Vision/Basic Container Operations/F_VN_SetAt/F_VN_SetAt_ULINT', node_F_VN_SetAt_ULINT);
NodeFactory.AddNodeAsPrototype('Vision/Basic Container Operations/F_VN_SetAt/F_VN_SetAt_USINT', node_F_VN_SetAt_USINT);

//NodeFactory.AddNodeAsPrototype('Vision/Basic Container Operations/F_VN_AdvanceIterator', node_F_VN_AdvanceIterator);
NodeFactory.AddNodeAsPrototype('Vision/Basic Container Operations/F_VN_CheckIfEmpty', node_F_VN_CheckIfEmpty);
//NodeFactory.AddNodeAsPrototype('Vision/Basic Container Operations/F_VN_CheckIfIteratorIsAtEnd', node_F_VN_CheckIfIteratorIsAtEnd);
//NodeFactory.AddNodeAsPrototype('Vision/Basic Container Operations/F_VN_ConvertContainerType', node_F_VN_ConvertContainerType);
NodeFactory.AddNodeAsPrototype('Vision/Basic Container Operations/F_VN_CopyContainer', node_F_VN_CopyContainer);
//NodeFactory.AddNodeAsPrototype('Vision/Basic Container Operations/F_VN_CopyContainerElementsConditional_ITcVnContainer', node_F_VN_CopyContainerElementsConditional_ITcVnContainer);
//NodeFactory.AddNodeAsPrototype('Vision/Basic Container Operations/F_VN_CopyContainerElementsConditional_ITcVnForwardIterator', node_F_VN_CopyContainerElementsConditional_ITcVnForwardIterator);
NodeFactory.AddNodeAsPrototype('Vision/Basic Container Operations/F_VN_CreateContainer', node_F_VN_CreateContainer);
//NodeFactory.AddNodeAsPrototype('Vision/Basic Container Operations/F_VN_CreateContainerFromArray', node_F_VN_CreateContainerFromArray);
//NodeFactory.AddNodeAsPrototype('Vision/Basic Container Operations/F_VN_EraseFromContainer', node_F_VN_EraseFromContainer);
//NodeFactory.AddNodeAsPrototype('Vision/Basic Container Operations/F_VN_ExportContainer', node_F_VN_ExportContainer);
NodeFactory.AddNodeAsPrototype('Vision/Basic Container Operations/F_VN_ExportContainer_String', node_F_VN_ExportContainer_String);
//NodeFactory.AddNodeAsPrototype('Vision/Basic Container Operations/F_VN_ExportContainerSize', node_F_VN_ExportContainerSize);
//NodeFactory.AddNodeAsPrototype('Vision/Basic Container Operations/F_VN_ExportSubContainer', node_F_VN_ExportSubContainer);
NodeFactory.AddNodeAsPrototype('Vision/Basic Container Operations/F_VN_ExportSubContainer_String', node_F_VN_ExportSubContainer_String);
//NodeFactory.AddNodeAsPrototype('Vision/Basic Container Operations/F_VN_ExportSubContainerSize', node_F_VN_ExportSubContainerSize);
NodeFactory.AddNodeAsPrototype('Vision/Basic Container Operations/F_VN_ExtractContainerRange', node_F_VN_ExtractContainerRange);
//NodeFactory.AddNodeAsPrototype('Vision/Basic Container Operations/F_VN_GetContainer', node_F_VN_GetContainer);
//NodeFactory.AddNodeAsPrototype('Vision/Basic Container Operations/F_VN_GetContainerExp', node_F_VN_GetContainerExp);
//NodeFactory.AddNodeAsPrototype('Vision/Basic Container Operations/F_VN_GetForwardIterator', node_F_VN_GetForwardIterator);
NodeFactory.AddNodeAsPrototype('Vision/Basic Container Operations/F_VN_GetNumberOfElements', node_F_VN_GetNumberOfElements);
//NodeFactory.AddNodeAsPrototype('Vision/Basic Container Operations/F_VN_GetRandomAccessIterator', node_F_VN_GetRandomAccessIterator);
//NodeFactory.AddNodeAsPrototype('Vision/Basic Container Operations/F_VN_IncrementIterator', node_F_VN_IncrementIterator);
//NodeFactory.AddNodeAsPrototype('Vision/Basic Container Operations/F_VN_IteratorDistance', node_F_VN_IteratorDistance);
//NodeFactory.AddNodeAsPrototype('Vision/Basic Container Operations/F_VN_ReserveContainerMemory', node_F_VN_ReserveContainerMemory);
NodeFactory.AddNodeAsPrototype('Vision/Basic Container Operations/F_VN_ReverseContainer', node_F_VN_ReverseContainer);
//NodeFactory.AddNodeAsPrototype('Vision/Basic Container Operations/F_VN_SetContainer', node_F_VN_SetContainer);
//NodeFactory.AddNodeAsPrototype('Vision/Basic Container Operations/F_VN_SetIteratorToBegin', node_F_VN_SetIteratorToBegin);

// Basic Image Operations
//NodeFactory.AddNodeAsPrototype('Vision/Basic Image Operations/F_VN_CombineImageChannels', node_F_VN_CombineImageChannels);
NodeFactory.AddNodeAsPrototype('Vision/Basic Image Operations/F_VN_ConvertElementType', node_F_VN_ConvertElementType);
NodeFactory.AddNodeAsPrototype('Vision/Basic Image Operations/F_VN_ConvertElementTypeExp', node_F_VN_ConvertElementTypeExp);
NodeFactory.AddNodeAsPrototype('Vision/Basic Image Operations/F_VN_CopyImage', node_F_VN_CopyImage);
NodeFactory.AddNodeAsPrototype('Vision/Basic Image Operations/F_VN_CopyImageRegion', node_F_VN_CopyImageRegion);
NodeFactory.AddNodeAsPrototype('Vision/Basic Image Operations/F_VN_CopyImageRegionToRegion', node_F_VN_CopyImageRegionToRegion);
NodeFactory.AddNodeAsPrototype('Vision/Basic Image Operations/F_VN_CopyIntoDisplayableImage', node_F_VN_CopyIntoDisplayableImage);
NodeFactory.AddNodeAsPrototype('Vision/Basic Image Operations/F_VN_CreateAssociatedImage', node_F_VN_CreateAssociatedImage);
NodeFactory.AddNodeAsPrototype('Vision/Basic Image Operations/F_VN_CreateEmptyImage', node_F_VN_CreateEmptyImage);
NodeFactory.AddNodeAsPrototype('Vision/Basic Image Operations/F_VN_CreateImage', node_F_VN_CreateImage);
NodeFactory.AddNodeAsPrototype('Vision/Basic Image Operations/F_VN_CreateImageAndSetPixels', node_F_VN_CreateImageAndSetPixels);
//NodeFactory.AddNodeAsPrototype('Vision/Basic Image Operations/F_VN_CreateImageFromArray', node_F_VN_CreateImageFromArray);
//NodeFactory.AddNodeAsPrototype('Vision/Basic Image Operations/F_VN_ExportImage', node_F_VN_ExportImage);
//NodeFactory.AddNodeAsPrototype('Vision/Basic Image Operations/F_VN_ExportImageAsBmp', node_F_VN_ExportImageAsBmp);
//NodeFactory.AddNodeAsPrototype('Vision/Basic Image Operations/F_VN_ExportImageAsBmpExp', node_F_VN_ExportImageAsBmpExp);
NodeFactory.AddNodeAsPrototype('Vision/Basic Image Operations/F_VN_ExportImageAsBmpSize', node_F_VN_ExportImageAsBmpSize);
NodeFactory.AddNodeAsPrototype('Vision/Basic Image Operations/F_VN_ExportImageAsBmpSizeExp', node_F_VN_ExportImageAsBmpSizeExp);
NodeFactory.AddNodeAsPrototype('Vision/Basic Image Operations/F_VN_ExportImageSize', node_F_VN_ExportImageSize);
NodeFactory.AddNodeAsPrototype('Vision/Basic Image Operations/F_VN_FuseImages', node_F_VN_FuseImages);
//NodeFactory.AddNodeAsPrototype('Vision/Basic Image Operations/F_VN_FuseImagesArray', node_F_VN_FuseImagesArray);
NodeFactory.AddNodeAsPrototype('Vision/Basic Image Operations/F_VN_GetImageChannel', node_F_VN_GetImageChannel);
NodeFactory.AddNodeAsPrototype('Vision/Basic Image Operations/F_VN_GetImageHeight', node_F_VN_GetImageHeight);
NodeFactory.AddNodeAsPrototype('Vision/Basic Image Operations/F_VN_GetImageInfo', node_F_VN_GetImageInfo);
NodeFactory.AddNodeAsPrototype('Vision/Basic Image Operations/F_VN_GetImageWidth', node_F_VN_GetImageWidth);
NodeFactory.AddNodeAsPrototype('Vision/Basic Image Operations/F_VN_GetPixel', node_F_VN_GetPixel);
NodeFactory.AddNodeAsPrototype('Vision/Basic Image Operations/F_VN_GetPixelFormat', node_F_VN_GetPixelFormat);
NodeFactory.AddNodeAsPrototype('Vision/Basic Image Operations/F_VN_GetRoi', node_F_VN_GetRoi);
NodeFactory.AddNodeAsPrototype('Vision/Basic Image Operations/F_VN_MixImageChannels', node_F_VN_MixImageChannels);
NodeFactory.AddNodeAsPrototype('Vision/Basic Image Operations/F_VN_ResetRoi', node_F_VN_ResetRoi);
NodeFactory.AddNodeAsPrototype('Vision/Basic Image Operations/F_VN_SetImageChannel', node_F_VN_SetImageChannel);
NodeFactory.AddNodeAsPrototype('Vision/Basic Image Operations/F_VN_SetPixel', node_F_VN_SetPixel);
NodeFactory.AddNodeAsPrototype('Vision/Basic Image Operations/F_VN_SetPixels', node_F_VN_SetPixels);
NodeFactory.AddNodeAsPrototype('Vision/Basic Image Operations/F_VN_SetPixelsExp', node_F_VN_SetPixelsExp);
NodeFactory.AddNodeAsPrototype('Vision/Basic Image Operations/F_VN_SetRoi', node_F_VN_SetRoi);
NodeFactory.AddNodeAsPrototype('Vision/Basic Image Operations/F_VN_SetRoi_TcVnRectangle_DINT', node_F_VN_SetRoi_TcVnRectangle_DINT);
NodeFactory.AddNodeAsPrototype('Vision/Basic Image Operations/F_VN_SetRoi_TcVnRectangle_UDINT', node_F_VN_SetRoi_TcVnRectangle_UDINT);
//NodeFactory.AddNodeAsPrototype('Vision/Basic Image Operations/F_VN_SplitImageChannels, node_F_VN_SplitImageChannels);
NodeFactory.AddNodeAsPrototype('Vision/Basic Image Operations/F_VN_TransformIntoDisplayableImage', node_F_VN_TransformIntoDisplayableImage); 
NodeFactory.AddNodeAsPrototype('Vision/Basic Image Operations/F_VN_TransformIntoDisplayableImageExp', node_F_VN_TransformIntoDisplayableImageExp); 
NodeFactory.AddNodeAsPrototype('Vision/Basic Image Operations/F_VN_CreateNDimensionalImage', node_F_VN_CreateNDimensionalImage);
NodeFactory.AddNodeAsPrototype('Vision/Basic Image Operations/F_VN_CreateNDimensionalImageAndSetPixels', node_F_VN_CreateNDimensionalImageAndSetPixels);
//NodeFactory.AddNodeAsPrototype('Vision/Basic Image Operations/F_VN_CreateNDimensionalImageFromArray, node_F_VN_CreateNDimensionalImageFromArray);
NodeFactory.AddNodeAsPrototype('Vision/Basic Image Operations/F_VN_GetLayoutInfo', node_F_VN_GetLayoutInfo);
NodeFactory.AddNodeAsPrototype('Vision/Basic Image Operations/F_VN_PadImageBorder', node_F_VN_PadImageBorder);
NodeFactory.AddNodeAsPrototype('Vision/Basic Image Operations/F_VN_PadImageBorderExp', node_F_VN_PadImageBorderExp);
//NodeFactory.AddNodeAsPrototype('Vision/Basic Image Operations/F_VN_ReinterpretUnsupportedImage', node_F_VN_ReinterpretUnsupportedImage);

// Code Quality
NodeFactory.AddNodeAsPrototype('Vision/Code Quality/F_VN_GradeBarcode', node_F_VN_GradeBarcode);
NodeFactory.AddNodeAsPrototype('Vision/Code Quality/F_VN_GradeBarcodeExp', node_F_VN_GradeBarcodeExp);
NodeFactory.AddNodeAsPrototype('Vision/Code Quality/F_VN_GradeDataMatrixCode', node_F_VN_GradeDataMatrixCode);
NodeFactory.AddNodeAsPrototype('Vision/Code Quality/F_VN_GradeDataMatrixCodeExp', node_F_VN_GradeDataMatrixCodeExp);
NodeFactory.AddNodeAsPrototype('Vision/Code Quality/F_VN_GradeQRCode', node_F_VN_GradeQRCode);
NodeFactory.AddNodeAsPrototype('Vision/Code Quality/F_VN_GradeQRCodeExp', node_F_VN_GradeQRCodeExp);

// Code Reading
NodeFactory.AddNodeAsPrototype('Vision/Code Reading/F_VN_AnalyzeBarcodeWalsh', node_F_VN_AnalyzeBarcodeWalsh);
NodeFactory.AddNodeAsPrototype('Vision/Code Reading/F_VN_DetectBarcodesWalsh', node_F_VN_DetectBarcodesWalsh);
NodeFactory.AddNodeAsPrototype('Vision/Code Reading/F_VN_DetectCodesNeuralNetwork', node_F_VN_DetectCodesNeuralNetwork);
NodeFactory.AddNodeAsPrototype('Vision/Code Reading/F_VN_ReadBarcode', node_F_VN_ReadBarcode);
NodeFactory.AddNodeAsPrototype('Vision/Code Reading/F_VN_ReadBarcodeExp', node_F_VN_ReadBarcodeExp);
NodeFactory.AddNodeAsPrototype('Vision/Code Reading/F_VN_ReadBarcodeExp2', node_F_VN_ReadBarcodeExp2);
NodeFactory.AddNodeAsPrototype('Vision/Code Reading/F_VN_ReadBarcodeRoi', node_F_VN_ReadBarcodeRoi);
NodeFactory.AddNodeAsPrototype('Vision/Code Reading/F_VN_ReadBarcodeRoiExp', node_F_VN_ReadBarcodeRoiExp);
NodeFactory.AddNodeAsPrototype('Vision/Code Reading/F_VN_ReadDataMatrixCode', node_F_VN_ReadDataMatrixCode);
NodeFactory.AddNodeAsPrototype('Vision/Code Reading/F_VN_ReadDataMatrixCodeExp', node_F_VN_ReadDataMatrixCodeExp);
NodeFactory.AddNodeAsPrototype('Vision/Code Reading/F_VN_ReadDataMatrixCodeExp2', node_F_VN_ReadDataMatrixCodeExp2);
NodeFactory.AddNodeAsPrototype('Vision/Code Reading/F_VN_ReadDataMatrixCodeRoi', node_F_VN_ReadDataMatrixCodeRoi);
NodeFactory.AddNodeAsPrototype('Vision/Code Reading/F_VN_ReadDataMatrixCodeRoiExp', node_F_VN_ReadDataMatrixCodeRoiExp);
NodeFactory.AddNodeAsPrototype('Vision/Code Reading/F_VN_ReadDotCodeRoi', Node_F_VN_ReadDotCodeRoi);
NodeFactory.AddNodeAsPrototype('Vision/Code Reading/F_VN_ReadDotCodeRoiExp', Node_F_VN_ReadDotCodeRoiExp);
NodeFactory.AddNodeAsPrototype('Vision/Code Reading/F_VN_ReadPharmaCode', node_F_VN_ReadPharmaCode);
NodeFactory.AddNodeAsPrototype('Vision/Code Reading/F_VN_ReadPharmaCodeExp', node_F_VN_ReadPharmaCodeExp);
NodeFactory.AddNodeAsPrototype('Vision/Code Reading/F_VN_ReadPharmaCodeExp2', node_F_VN_ReadPharmaCodeExp2);
NodeFactory.AddNodeAsPrototype('Vision/Code Reading/F_VN_ReadQRCode', node_F_VN_ReadQRCode);
NodeFactory.AddNodeAsPrototype('Vision/Code Reading/F_VN_ReadQRCodeExp', node_F_VN_ReadQRCodeExp);
NodeFactory.AddNodeAsPrototype('Vision/Code Reading/F_VN_ReadQRCodeExp2', node_F_VN_ReadQRCodeExp2);

// Constants
NodeFactory.AddNodeAsPrototype('Vision/Constants/RGBA_BLACK', node_RGBA_BLACK);
NodeFactory.AddNodeAsPrototype('Vision/Constants/RGBA_RED', node_RGBA_RED);
NodeFactory.AddNodeAsPrototype('Vision/Constants/RGBA_YELLOW', node_RGBA_YELLOW);
NodeFactory.AddNodeAsPrototype('Vision/Constants/RGBA_GREEN', node_RGBA_GREEN);
NodeFactory.AddNodeAsPrototype('Vision/Constants/RGBA_CYAN', node_RGBA_CYAN);
NodeFactory.AddNodeAsPrototype('Vision/Constants/RGBA_BLUE', node_RGBA_BLUE);
NodeFactory.AddNodeAsPrototype('Vision/Constants/RGBA_MAGENTA', node_RGBA_MAGENTA);
NodeFactory.AddNodeAsPrototype('Vision/Constants/RGBA_WHITE', node_RGBA_WHITE);
NodeFactory.AddNodeAsPrototype('Vision/Constants/RGBA_RANDOM', node_RGBA_RANDOM);
NodeFactory.AddNodeAsPrototype('Vision/Constants/ContainerType_Vector_SINT', node_ContainerType_Vector_SINT);
NodeFactory.AddNodeAsPrototype('Vision/Constants/ContainerType_Vector_USINT', node_ContainerType_Vector_USINT);
NodeFactory.AddNodeAsPrototype('Vision/Constants/ContainerType_Vector_INT', node_ContainerType_Vector_INT);
NodeFactory.AddNodeAsPrototype('Vision/Constants/ContainerType_Vector_UINT', node_ContainerType_Vector_UINT);
NodeFactory.AddNodeAsPrototype('Vision/Constants/ContainerType_Vector_DINT', node_ContainerType_Vector_DINT);
NodeFactory.AddNodeAsPrototype('Vision/Constants/ContainerType_Vector_UDINT', node_ContainerType_Vector_UDINT);
NodeFactory.AddNodeAsPrototype('Vision/Constants/ContainerType_Vector_ULINT', node_ContainerType_Vector_ULINT);
NodeFactory.AddNodeAsPrototype('Vision/Constants/ContainerType_Vector_REAL', node_ContainerType_Vector_REAL);
NodeFactory.AddNodeAsPrototype('Vision/Constants/ContainerType_Vector_LREAL', node_ContainerType_Vector_LREAL);
NodeFactory.AddNodeAsPrototype('Vision/Constants/ContainerType_Vector_ITcVnImage', node_ContainerType_Vector_ITcVnImage);
NodeFactory.AddNodeAsPrototype('Vision/Constants/ContainerType_Vector_TcVnPoint2_DINT', node_ContainerType_Vector_TcVnPoint2_DINT);
NodeFactory.AddNodeAsPrototype('Vision/Constants/ContainerType_Vector_TcVnPoint2_REAL', node_ContainerType_Vector_TcVnPoint2_REAL);
NodeFactory.AddNodeAsPrototype('Vision/Constants/ContainerType_Vector_TcVnPoint2_LREAL', node_ContainerType_Vector_TcVnPoint2_LREAL);
NodeFactory.AddNodeAsPrototype('Vision/Constants/ContainerType_Vector_TcVnPoint3_REAL', node_ContainerType_Vector_TcVnPoint3_REAL);
NodeFactory.AddNodeAsPrototype('Vision/Constants/ContainerType_Vector_TcVnPoint3_LREAL', node_ContainerType_Vector_TcVnPoint3_LREAL);
NodeFactory.AddNodeAsPrototype('Vision/Constants/ContainerType_Vector_Vector_TcVnPoint2_DINT', node_ContainerType_Vector_Vector_TcVnPoint2_DINT);
NodeFactory.AddNodeAsPrototype('Vision/Constants/ContainerType_Vector_Vector_TcVnPoint2_REAL', node_ContainerType_Vector_Vector_TcVnPoint2_REAL);
NodeFactory.AddNodeAsPrototype('Vision/Constants/ContainerType_Vector_Vector_TcVnPoint3_REAL', node_ContainerType_Vector_Vector_TcVnPoint3_REAL);
NodeFactory.AddNodeAsPrototype('Vision/Constants/ContainerType_Vector_Vector_UDINT', node_ContainerType_Vector_Vector_UDINT);
NodeFactory.AddNodeAsPrototype('Vision/Constants/ContainerType_Vector_Vector_ULINT', node_ContainerType_Vector_Vector_ULINT);
NodeFactory.AddNodeAsPrototype('Vision/Constants/ContainerType_Vector_Vector_REAL', node_ContainerType_Vector_Vector_REAL);
NodeFactory.AddNodeAsPrototype('Vision/Constants/ContainerType_Vector_Vector_LREAL', node_ContainerType_Vector_Vector_LREAL);
NodeFactory.AddNodeAsPrototype('Vision/Constants/ContainerType_Vector_TcVnVector2_SINT', node_ContainerType_Vector_TcVnVector2_SINT);
NodeFactory.AddNodeAsPrototype('Vision/Constants/ContainerType_Vector_TcVnVector2_USINT', node_ContainerType_Vector_TcVnVector2_USINT);
NodeFactory.AddNodeAsPrototype('Vision/Constants/ContainerType_Vector_TcVnVector2_INT', node_ContainerType_Vector_TcVnVector2_INT);
NodeFactory.AddNodeAsPrototype('Vision/Constants/ContainerType_Vector_TcVnVector2_UINT', node_ContainerType_Vector_TcVnVector2_UINT);
NodeFactory.AddNodeAsPrototype('Vision/Constants/ContainerType_Vector_TcVnVector2_DINT', node_ContainerType_Vector_TcVnVector2_DINT);
NodeFactory.AddNodeAsPrototype('Vision/Constants/ContainerType_Vector_TcVnVector2_REAL', node_ContainerType_Vector_TcVnVector2_REAL);
NodeFactory.AddNodeAsPrototype('Vision/Constants/ContainerType_Vector_TcVnVector3_SINT', node_ContainerType_Vector_TcVnVector3_SINT);
NodeFactory.AddNodeAsPrototype('Vision/Constants/ContainerType_Vector_TcVnVector3_USINT', node_ContainerType_Vector_TcVnVector3_USINT);
NodeFactory.AddNodeAsPrototype('Vision/Constants/ContainerType_Vector_TcVnVector3_INT', node_ContainerType_Vector_TcVnVector3_INT);
NodeFactory.AddNodeAsPrototype('Vision/Constants/ContainerType_Vector_TcVnVector3_UINT', node_ContainerType_Vector_TcVnVector3_UINT);
NodeFactory.AddNodeAsPrototype('Vision/Constants/ContainerType_Vector_TcVnVector3_REAL', node_ContainerType_Vector_TcVnVector3_REAL);
NodeFactory.AddNodeAsPrototype('Vision/Constants/ContainerType_Vector_TcVnVector4_SINT', node_ContainerType_Vector_TcVnVector4_SINT);
NodeFactory.AddNodeAsPrototype('Vision/Constants/ContainerType_Vector_TcVnVector4_USINT', node_ContainerType_Vector_TcVnVector4_USINT);
NodeFactory.AddNodeAsPrototype('Vision/Constants/ContainerType_Vector_TcVnVector4_INT', node_ContainerType_Vector_TcVnVector4_INT);
NodeFactory.AddNodeAsPrototype('Vision/Constants/ContainerType_Vector_TcVnVector4_UINT', node_ContainerType_Vector_TcVnVector4_UINT);
NodeFactory.AddNodeAsPrototype('Vision/Constants/ContainerType_Vector_TcVnVector4_DINT', node_ContainerType_Vector_TcVnVector4_DINT);
NodeFactory.AddNodeAsPrototype('Vision/Constants/ContainerType_Vector_TcVnVector4_REAL', node_ContainerType_Vector_TcVnVector4_REAL);
NodeFactory.AddNodeAsPrototype('Vision/Constants/ContainerType_Vector_TcVnVector4_LREAL', node_ContainerType_Vector_TcVnVector4_LREAL);
NodeFactory.AddNodeAsPrototype('Vision/Constants/ContainerType_Vector_TcVnRectangle_DINT', node_ContainerType_Vector_TcVnRectangle_DINT);
NodeFactory.AddNodeAsPrototype('Vision/Constants/ContainerType_Vector_TcVnRotatedRectangle', node_ContainerType_Vector_TcVnRotatedRectangle);
NodeFactory.AddNodeAsPrototype('Vision/Constants/ContainerType_Vector_TcVnKeyPoint', node_ContainerType_Vector_TcVnKeyPoint);
NodeFactory.AddNodeAsPrototype('Vision/Constants/ContainerType_Vector_TcVnDMatch', node_ContainerType_Vector_TcVnDMatch);
NodeFactory.AddNodeAsPrototype('Vision/Constants/ContainerType_Vector_Vector_TcVnDMatch', node_ContainerType_Vector_Vector_TcVnDMatch);
NodeFactory.AddNodeAsPrototype('Vision/Constants/ContainerType_String_SINT', node_ContainerType_String_SINT);
NodeFactory.AddNodeAsPrototype('Vision/Constants/ContainerType_Vector_String_SINT', node_ContainerType_Vector_String_SINT);

